FUNCTION_BLOCK "FB_PowerOn"   // FB462, SCL
{ S7_Optimized_Access := 'TRUE' }
// stored: AutoNumber false, MemoryReserve 100, SetENOAutomatically false
   VAR
      sMachinePower : Bool;
      sMachineReadySoft : Bool;
      sOkForPowerON : Bool;
      sTimeMachineReadyDelay { S7_SetPoint := 'True'} : TON_TIME;
      sDelayPowerOFF { S7_SetPoint := 'True'} : TON_TIME;
      sDelayPowerON_1 { S7_SetPoint := 'True'} : TON_TIME;
      sDelayPowerON_2 { S7_SetPoint := 'True'} : TON_TIME;
      sX_AxisBrakeRelease { S7_SetPoint := 'True'} : Bool;
      sY_AxisBrakeRelease : Bool;
      sB_AxisBrakeRelease : Bool;
   END_VAR
   VAR CONSTANT
      TIME_MACHINE_IN_DELAY : Time := T#2S;   // Output short pulse blinking
   END_VAR
BEGIN
   REGION Description header 
       //==================================================================================
       // POSALUX Swiss SA / (C) Copyright 2024
       //----------------------------------------------------------------------------------
       // Title: Power de la machine
       // Comment/Function: 
       //  A revoir le power des differents elements
       // Author: Gowsigan SRITHARAN
       // Engineering: TIA Portal v17
       //----------------------------------------------------------------------------------
       // Change log table:
       // Version  | Date     | Expert in charge | Changes applied
       // ---------|----------|------------------|------------------------------------
       // 00.00.01 | 20241120 | GSR              | First released version
       // ==================================================================================
   END_REGION

   REGION General Circuit breaker
       IF NOT "DB_DigitalInputs".sBreakerCtrl.sSWStatus THEN
           "LBP_AlarmMsgs".UserA[0].A70UUxx[3] := TRUE;
       END_IF;
   END_REGION

   REGION Operating counter
       "DB_DigitalOutputs".sOperatingCounter.sSWStatus :=
       ("LBP_Chan1".E_ProgRunning
       OR "LBP_Chan1".E_ProgWait)
       AND "LBP_ModeGroup".E_AUTO;
   END_REGION

   REGION Axis power requested
       #sOkForPowerON := "LBP_NC".E_NCKready AND "LBP_NC".E_DrivesInCylOp AND "DB_DataFromSafety".EmergencyStop AND NOT "DB_Alarms".sAlarmsLevel5 AND NOT "DB_Alarms".sAlarmsLevel6;

       IF #sOkForPowerON AND "DB_McpKeyboardSignals".sPowerON.sKeySWPositiveFront THEN
           #sMachinePower := TRUE;
       END_IF;

       IF  "DB_McpKeyboardSignals".sPowerOFF.sKeySWNegativeFront
           OR "DB_Machineshutdown_UPS".sShutDownPower
           OR "DB_Alarms".sAlarmsLevel5
           OR NOT "DB_DataFromSafety".EmergencyStop THEN
           #sMachinePower := FALSE;
       END_IF;

   END_REGION

   REGION Axis power output and waiting machine ready
       #sDelayPowerOFF(IN := NOT "LBP_NC".E_611Dready AND NOT #sMachinePower,
                       PT := T#1s);

       #sDelayPowerON_1(IN := "DB_DigitalOutputs".sInfeedON.sSWStatus,
                        PT := t#2s);
       #sDelayPowerON_2(IN := "DB_DigitalOutputs".sAxisActivation.sSWStatus,
                        PT := t#2s);
       IF #sMachinePower THEN
           "DB_DigitalOutputs".sInfeedON.sSWStatus := TRUE;
           IF #sDelayPowerON_1.Q THEN
               "DB_DigitalOutputs".sAxisActivation.sSWStatus := TRUE;
           END_IF;
           IF #sDelayPowerON_2.Q THEN

               "DB_DigitalOutputs".sAxis2_PowerContactor.sSWStatus  := TRUE;
               "DB_DigitalOutputs".sXY_AxisPowerContactor.sSWStatus := TRUE;
               "DB_DigitalOutputs".sBus60V_PowerContactor.sSWStatus := TRUE;
           END_IF;
       ELSE
           "DB_DigitalOutputs".sAxisActivation.sSWStatus := FALSE;

           IF #sDelayPowerOFF.Q THEN
               "DB_DigitalOutputs".sAxis2_PowerContactor.sSWStatus  := FALSE;
               "DB_DigitalOutputs".sXY_AxisPowerContactor.sSWStatus := FALSE;
               "DB_DigitalOutputs".sBus60V_PowerContactor.sSWStatus := FALSE;
               "DB_DigitalOutputs".sInfeedON.sSWStatus := FALSE;
           END_IF;
       END_IF;

       #sMachineReadySoft := "LBP_NC".E_611Dready;
   END_REGION

   REGION Machine in delay
       #sTimeMachineReadyDelay.TON(IN := #sMachineReadySoft,
                                   PT := #TIME_MACHINE_IN_DELAY);
   END_REGION

   REGION LED Machine ready start
       "DB_McpKeyboardSignals".sPowerON.sLedSWStatus :=
       (NOT #sMachinePower AND #sOkForPowerON AND "Clock_0.5Hz")
       OR (NOT #sTimeMachineReadyDelay.Q AND #sMachinePower AND "Clock_2Hz")
       OR #sTimeMachineReadyDelay.Q AND #sMachineReadySoft;
   END_REGION

   REGION Axis Brake
       // X Axis Brake Activation
       "DB_DigitalOutputs".sX_AxisBrakeActivation.sSWStatus := (("LBP_Axis01_X".E_AxisReady
       AND "LBP_Axis01_X".E_MotOK
       AND "LBP_Axis01_X".E_PulseEnable)
       OR #sX_AxisBrakeRelease);

       // Y Axis Brake Activation    
       "DB_DigitalOutputs".sY_AxisBrakeActivation.sSWStatus := (("LBP_Axis02_Y".E_AxisReady
       AND "LBP_Axis02_Y".E_MotOK
       AND "LBP_Axis02_Y".E_PulseEnable)
       OR #sY_AxisBrakeRelease);

       // B Axis Brake Activation   
       "DB_DigitalOutputs".sB_AxisBrakeRelease.sSWStatus := ("LBP_Axis04_B".E_AxisReady
       AND "LBP_Axis05_U1".E_MotOK
       AND "LBP_Axis05_U1".E_PulseEnable)
       OR #sB_AxisBrakeRelease;

       // Axis feed stop
       "LBP_AlarmMsgs".AxisA[1].AAFdStop60AAxx[0] := NOT "DB_DigitalOutputs".sX_AxisBrakeActivation.sSWStatus;     // X Axis
       "LBP_AlarmMsgs".AxisA[2].AAFdStop60AAxx[0] := NOT "DB_DigitalOutputs".sY_AxisBrakeActivation.sSWStatus;     // Y Axis
       "LBP_AlarmMsgs".AxisA[4].AAFdStop60AAxx[0] := NOT "DB_DigitalOutputs".sB_AxisBrakeRelease.sSWStatus;        // B Axis
   END_REGION
END_FUNCTION_BLOCK

FUNCTION_BLOCK "FB_Maintenances"   // FB473, SCL
{ S7_Optimized_Access := 'TRUE' }
// stored: AutoNumber false, MemoryReserve 100, SetENOAutomatically false
   VAR
      sCheckMachine : "FB_Maintenance";   // Message: Check Laser optical path (84h)
      sReplaceAirConditioningFilter { S7_SetPoint := 'True'} : "FB_Maintenance";   // Message: Clean the fairing (200 h)
      sMachineCooling_ReplaceWaterFilter { S7_SetPoint := 'True'} : "FB_Maintenance";   // Message: Clean the sheet metal (200 h)
      sTermotekChiller_ChangeFilterAndWater { S7_SetPoint := 'True'} : "FB_Maintenance";   // Message: Clean the screens (200 h)
      sCheckSafetySystem { S7_SetPoint := 'True'} : "FB_Maintenance";   // Message: Check the machine (200 h)
      sReplaceTipShellPeekGripper { S7_SetPoint := 'True'} : "FB_Maintenance";   // Message: Clean the clamping (200 h)
      sReplaceFiltersVacuumLoadingUnloading { S7_SetPoint := 'True'} : "FB_Maintenance";   // Message: Check the filter of the Laser power unit (2000 h)
      sReplaceFiltersVacuumGenerator { S7_SetPoint := 'True'} : "FB_Maintenance";   // Message: Check the safety systems (2000 h)
      sReplaceFilterAirDryer { S7_SetPoint := 'True'} : "FB_Maintenance";   // Message: Grease the X axis (1 y)
      sReplace5umFilter { S7_SetPoint := 'True'} : "FB_Maintenance";   // Message: Grease the Y axis (1 y)
      sReplace01umFilter { S7_SetPoint := 'True'} : "FB_Maintenance";   // Message: Check the water level of the TERMOTEK cooler (24 h)
      sReplaceActiveCarbonFilter { S7_SetPoint := 'True'} : "FB_Maintenance";   // Message: Clean the grid of the TERMOTEK cooler (24 h)
      sUTLExtraction_ReplaceParticleFilter { S7_SetPoint := 'True'} : "FB_Maintenance";   // Message: Check the operation of the condensate drain (24 h)
      sUTLExtraction_ReplaceFilterCassetteAndActiveCarbonFilter { S7_SetPoint := 'True'} : "FB_Maintenance";   // Message: Check the dew point under pressure (24 h)
      sReplaceSealOnSas { S7_SetPoint := 'True'} : "FB_Maintenance";   // Message: Clean the grid of the air dryer (24 h)
      sGreaseAxes { S7_SetPoint := 'True'} : "FB_Maintenance";   // Message: Replace the line filter of the air dryer (600 h)
      sMaintenance_16 { S7_SetPoint := 'True'} : "FB_Maintenance";   // Message: Replace 5 µm filter cartridge (600 h)
      sMaintenance_17 { S7_SetPoint := 'True'} : "FB_Maintenance";   // Message: Replace 0.01 µm filter cartridge (600 h)
      sMaintenance_18 { S7_SetPoint := 'True'} : "FB_Maintenance";   // Message: Replace the particles filter of the suction system (1000 h)
      sMaintenance_19 { S7_SetPoint := 'True'} : "FB_Maintenance";   // Message: Replace the filtration cassette AND the actived carbon of the suction system (1000 h)
      sMaintenance_20 { S7_SetPoint := 'True'} : "FB_Maintenance";   // Message: Replace the air conditioning filter (1000 h)
      sMaintenance_21 { S7_SetPoint := 'True'} : "FB_Maintenance";   // Message: Replace the TERMOTEK cooler filter (2000 h)
      sMaintenance_22 { S7_SetPoint := 'True'} : "FB_Maintenance";   // Message: Replace the water of the TERMOTEK cooler (2000 h)
      sMaintenance_23 { S7_SetPoint := 'True'} : "FB_Maintenance";   // Message: Spare
      sMaintenance_24 { S7_SetPoint := 'True'} : "FB_Maintenance";   // Message: Spare
      sMaintenance_25 { S7_SetPoint := 'True'} : "FB_Maintenance";   // Message: Spare
      sMaintenance_26 { S7_SetPoint := 'True'} : "FB_Maintenance";   // Message: Spare
      sMaintenance_27 { S7_SetPoint := 'True'} : "FB_Maintenance";   // Message: Spare
      sMaintenance_28 { S7_SetPoint := 'True'} : "FB_Maintenance";   // Message: Spare
      sMaintenance_29 { S7_SetPoint := 'True'} : "FB_Maintenance";   // Message: Spare
      sMaintenance_30 { S7_SetPoint := 'True'} : "FB_Maintenance";   // Message: Spare
      sMaintenance_31 { S7_SetPoint := 'True'} : "FB_Maintenance";   // Message: Spare
      sMaintenance_32 { S7_SetPoint := 'True'} : "FB_Maintenance";   // Message: Spare
      sMaintenance_33 { S7_SetPoint := 'True'} : "FB_Maintenance";   // Message: Spare
      sMaintenance_34 { S7_SetPoint := 'True'} : "FB_Maintenance";   // Message: Spare
      sMaintenance_35 { S7_SetPoint := 'True'} : "FB_Maintenance";   // Message: Spare
      sMaintenance_36 { S7_SetPoint := 'True'} : "FB_Maintenance";   // Message: Spare
      sMaintenance_37 { S7_SetPoint := 'True'} : "FB_Maintenance";   // Message: Spare
      sMaintenance_38 { S7_SetPoint := 'True'} : "FB_Maintenance";   // Message: Spare
      sMaintenance_39 { S7_SetPoint := 'True'} : "FB_Maintenance";   // Message: Spare
      sMaintenance_40 { S7_SetPoint := 'True'} : "FB_Maintenance";   // Message: Spare
      sMaintenance_41 { S7_SetPoint := 'True'} : "FB_Maintenance";   // Message: Spare
      sMaintenance_42 { S7_SetPoint := 'True'} : "FB_Maintenance";   // Message: Spare
      sMaintenance_43 { S7_SetPoint := 'True'} : "FB_Maintenance";   // Message: Spare
      sMaintenance_44 { S7_SetPoint := 'True'} : "FB_Maintenance";   // Message: Spare
      sMaintenance_45 { S7_SetPoint := 'True'} : "FB_Maintenance";   // Message: Spare
      sMaintenance_46 { S7_SetPoint := 'True'} : "FB_Maintenance";   // Message: Spare
      sMaintenance_47 { S7_SetPoint := 'True'} : "FB_Maintenance";   // Message: Spare
      sMaintenance_48 { S7_SetPoint := 'True'} : "FB_Maintenance";   // Message: Spare
      sMaintenance_49 { S7_SetPoint := 'True'} : "FB_Maintenance";   // Message: Spare
      sMaintenance_50 { S7_SetPoint := 'True'} : "FB_Maintenance";   // Message: Spare
      sMaintenance_51 { S7_SetPoint := 'True'} : "FB_Maintenance";   // Message: Spare
      sMaintenance_52 { S7_SetPoint := 'True'} : "FB_Maintenance";   // Message: Spare
      sMaintenance_53 { S7_SetPoint := 'True'} : "FB_Maintenance";   // Message: Spare
      sMaintenance_54 { S7_SetPoint := 'True'} : "FB_Maintenance";   // Message: Spare
      sMaintenance_55 { S7_SetPoint := 'True'} : "FB_Maintenance";   // Message: Spare
      sMaintenance_56 { S7_SetPoint := 'True'} : "FB_Maintenance";   // Message: Spare
      sMaintenance_57 { S7_SetPoint := 'True'} : "FB_Maintenance";   // Message: Spare
      sMaintenance_58 { S7_SetPoint := 'True'} : "FB_Maintenance";   // Message: Spare
      sMaintenance_59 { S7_SetPoint := 'True'} : "FB_Maintenance";   // Message: Spare
      sMaintenance_60 { S7_SetPoint := 'True'} : "FB_Maintenance";   // Message: Spare
      sMaintenance_61 { S7_SetPoint := 'True'} : "FB_Maintenance";   // Message: Spare
      sMaintenance_62 { S7_SetPoint := 'True'} : "FB_Maintenance";   // Message: Spare
      sMaintenance_63 { S7_SetPoint := 'True'} : "FB_Maintenance";   // Message: Spare
   END_VAR
BEGIN
   REGION Description header 
       //==================================================================================
       // POSALUX Swiss SA / (C) Copyright 2024
       //----------------------------------------------------------------------------------
       // Title: Maintenance
       // Comment/Function: Liste des apparaeils à controler dans la Liste des équipements 
       //                   pour la maintenance préventive  
       //
       // Author: Gowsigan SRITHARAN
       // Engineering: TIA Portal v17
       //----------------------------------------------------------------------------------
       // Change log table:
       // Version  | Date     | Expert in charge | Changes applied
       // ---------|----------|------------------|------------------------------------
       // 00.00.01 | 20250912 | WFA              | First released version
       // ==================================================================================
   END_REGION

   REGION 200 hours
           // Check the machine
           #sCheckMachine(iIncrementEnable := "LBP_Chan1".E_ProgRunning,
                          iID := 101,
                          ioOPC := "DB_OPC_Maintenance".Tasks[1],
                          ioAlarm := "LBP_AlarmMsgs".UserA[30].A70UUxx[00],
                          ioWarning := "LBP_AlarmMsgs".UserA[30].A70UUxx[32]);
      END_REGION

      REGION 1000 hours
           // Replace the air conditioning filter
           #sReplaceAirConditioningFilter(iIncrementEnable := "LBP_Chan1".E_ProgRunning,
                                          iID := 201,
                                          ioOPC := "DB_OPC_Maintenance".Tasks[2],
                                          ioAlarm := "LBP_AlarmMsgs".UserA[30].A70UUxx[01],
                                          ioWarning := "LBP_AlarmMsgs".UserA[30].A70UUxx[33]);

           // Machine cooling: replace water filter
           #sMachineCooling_ReplaceWaterFilter(iIncrementEnable := "LBP_Chan1".E_ProgRunning,
                                               iID := 202,
                                               ioOPC := "DB_OPC_Maintenance".Tasks[3],
                                               ioAlarm := "LBP_AlarmMsgs".UserA[30].A70UUxx[02],
                                               ioWarning := "LBP_AlarmMsgs".UserA[30].A70UUxx[34]);
      END_REGION

      REGION 2000 hours
          // Termotek chiller: change filter and water
          #sTermotekChiller_ChangeFilterAndWater(iIncrementEnable := "LBP_Chan1".E_ProgRunning,
                                                 iID := 301,
                                                 ioOPC := "DB_OPC_Maintenance".Tasks[4],
                                                 ioAlarm := "LBP_AlarmMsgs".UserA[30].A70UUxx[03],
                                                 ioWarning := "LBP_AlarmMsgs".UserA[30].A70UUxx[35]);

           // Check the safety system
           #sCheckSafetySystem(iIncrementEnable := "LBP_Chan1".E_ProgRunning,
                               iID := 302,
                               ioOPC := "DB_OPC_Maintenance".Tasks[5],
                               ioAlarm := "LBP_AlarmMsgs".UserA[30].A70UUxx[04],
                               ioWarning := "LBP_AlarmMsgs".UserA[30].A70UUxx[36]);

           // Replace the tip-shell PEEK gripper
           #sReplaceTipShellPeekGripper(iIncrementEnable := "LBP_Chan1".E_ProgRunning,
                                        iID := 303,
                                        ioOPC := "DB_OPC_Maintenance".Tasks[6],
                                        ioAlarm := "LBP_AlarmMsgs".UserA[30].A70UUxx[05],
                                        ioWarning := "LBP_AlarmMsgs".UserA[30].A70UUxx[37]);
      END_REGION

      REGION 3000 hours
           // Replace the filters for the vacuum of the loading/unloading
           #sReplaceFiltersVacuumLoadingUnloading(iIncrementEnable := "LBP_Chan1".E_ProgRunning,
                                                  iID := 401,
                                                  ioOPC := "DB_OPC_Maintenance".Tasks[7],
                                                  ioAlarm := "LBP_AlarmMsgs".UserA[30].A70UUxx[06],
                                                  ioWarning := "LBP_AlarmMsgs".UserA[30].A70UUxx[38]);

           // Replace the filters of the vacuum generator VADM
           #sReplaceFiltersVacuumGenerator(iIncrementEnable := "LBP_Chan1".E_ProgRunning,
                                           iID := 402,
                                           ioOPC := "DB_OPC_Maintenance".Tasks[8],
                                           ioAlarm := "LBP_AlarmMsgs".UserA[30].A70UUxx[07],
                                           ioWarning := "LBP_AlarmMsgs".UserA[30].A70UUxx[39]);
      END_REGION

      REGION 4000 hours
           // Replace the fine filter of the air dryer
           #sReplaceFilterAirDryer(iIncrementEnable := "LBP_Chan1".E_ProgRunning,
                                   iID := 501,
                                   ioOPC := "DB_OPC_Maintenance".Tasks[9],
                                   ioAlarm := "LBP_AlarmMsgs".UserA[30].A70UUxx[08],
                                   ioWarning := "LBP_AlarmMsgs".UserA[30].A70UUxx[40]);

           // Replace the 5 μm filter
           #sReplace5umFilter(iIncrementEnable := "LBP_Chan1".E_ProgRunning,
                              iID := 502,
                              ioOPC := "DB_OPC_Maintenance".Tasks[10],
                              ioAlarm := "LBP_AlarmMsgs".UserA[30].A70UUxx[09],
                              ioWarning := "LBP_AlarmMsgs".UserA[30].A70UUxx[41]);

          // Replace the 0.1 μm filter
         #sReplace01umFilter(iIncrementEnable := "LBP_Chan1".E_ProgRunning,
                             iID := 503,
                             ioOPC := "DB_OPC_Maintenance".Tasks[11],
                             ioAlarm := "LBP_AlarmMsgs".UserA[30].A70UUxx[10],
                             ioWarning := "LBP_AlarmMsgs".UserA[30].A70UUxx[42]);

           // Replace the active carbon filter
           #sReplaceActiveCarbonFilter(iIncrementEnable := "LBP_Chan1".E_ProgRunning,
                                       iID := 504,
                                       ioOPC := "DB_OPC_Maintenance".Tasks[12],
                                       ioAlarm := "LBP_AlarmMsgs".UserA[30].A70UUxx[11],
                                       ioWarning := "LBP_AlarmMsgs".UserA[30].A70UUxx[43]);

           // UTL extraction: replace particle filter
           #sUTLExtraction_ReplaceParticleFilter(iIncrementEnable := "LBP_Chan1".E_ProgRunning,
                                                 iID := 505,
                                                 ioOPC := "DB_OPC_Maintenance".Tasks[13],
                                                 ioAlarm := "LBP_AlarmMsgs".UserA[30].A70UUxx[12],
                                                 ioWarning := "LBP_AlarmMsgs".UserA[30].A70UUxx[44]);

           // UTL extraction: replace filter cassette and active carbon filter
           #sUTLExtraction_ReplaceFilterCassetteAndActiveCarbonFilter(iIncrementEnable := "LBP_Chan1".E_ProgRunning,
                                                                      iID := 506,
                                                                      ioOPC := "DB_OPC_Maintenance".Tasks[14],
                                                                      ioAlarm := "LBP_AlarmMsgs".UserA[30].A70UUxx[13],
                                                                      ioWarning := "LBP_AlarmMsgs".UserA[30].A70UUxx[45]);

      END_REGION

      REGION 6000 hours
           // Replace the seal on the air lock door (SAS)
           #sReplaceSealOnSas(iIncrementEnable := "LBP_Chan1".E_ProgRunning,
                              iID := 601,
                              ioOPC := "DB_OPC_Maintenance".Tasks[15],
                              ioAlarm := "LBP_AlarmMsgs".UserA[30].A70UUxx[14],
                              ioWarning := "LBP_AlarmMsgs".UserA[30].A70UUxx[46]);

           // Grease the axes
           #sGreaseAxes(iIncrementEnable := "LBP_Chan1".E_ProgRunning,
                        iID := 602,
                        ioOPC := "DB_OPC_Maintenance".Tasks[16],
                        ioAlarm := "LBP_AlarmMsgs".UserA[30].A70UUxx[15],
                        ioWarning := "LBP_AlarmMsgs".UserA[30].A70UUxx[47]);
      END_REGION
END_FUNCTION_BLOCK

FUNCTION_BLOCK "FB_Maintenance"   // FB471, SCL
{ S7_Optimized_Access := 'TRUE' }
// stored: AutoNumber false, MemoryReserve 100, SetENOAutomatically false
   VAR_INPUT
      iIncrementEnable { ExternalAccessible := 'False'; ExternalVisible := 'False'; ExternalWritable := 'False'} : Bool;
      iID { ExternalAccessible := 'False'; ExternalVisible := 'False'; ExternalWritable := 'False'} : Int;
   END_VAR
   VAR_IN_OUT
      ioOPC : "UDT_OPC_Maintenance";
      ioAlarm { ExternalAccessible := 'False'; ExternalVisible := 'False'; ExternalWritable := 'False'} : Bool;   // Alarme (100% atteint)
      ioWarning { ExternalAccessible := 'False'; ExternalVisible := 'False'; ExternalWritable := 'False'} : Bool;   // Avertissement (80% atteint)
   END_VAR
   VAR
      sElement { ExternalAccessible := 'False'; ExternalVisible := 'False'; ExternalWritable := 'False'} : "UDT_MaintenanceElement";
   END_VAR
   VAR_TEMP
      tUsagePercent : Real;
      tAdjustedIncrement : Bool;
   END_VAR
BEGIN
   REGION Description header 
       //==================================================================================
       // POSALUX Swiss SA / (C) Copyright 2024
       //----------------------------------------------------------------------------------
       // Title: Gestion_Temps_Fonctionnement
       // Comment/Function: Cette fonction  assure le suivi du temps de fonctionnement
       //                   des équipements et génère des alertes basées sur
       //                   leur utilisation. Elle incrémente le temps de fonctionnement
       //                   selon l'unité définie (minute, heure, jour), calcule le
       //                   pourcentage d'utilisation par rapport à un seuil d'alarme, et
       //                   gère les avertissements et alarmes en fonction de ce pourcentage
       //
       // Author: Gowsigan SRITHARAN
       // Engineering: TIA Portal v17
       //----------------------------------------------------------------------------------
       // Change log table:
       // Version  | Date     | Expert in charge | Changes applied
       // ---------|----------|------------------|------------------------------------
       // 00.00.01 | 20241120 | GSR              | First released version
       // ---------|----------|------------------|------------------------------------
       // 01.01.01 | 20241219 | FMI              | Utilisation d'un flanc montant du clock1Hz pour compter en secondes
       // ==================================================================================
   END_REGION

   REGION Incrementation du temps en secondes
       IF "DB_Impulsion".sRT_Clock_1Hz.Q AND #iIncrementEnable THEN
           #sElement.RunTimeSec := #sElement.RunTimeSec + 1;
       END_IF;
   END_REGION

   REGION Incrementation du temps en fonction du type unité
       CASE #sElement.TimeUnit OF
           0:
               #sElement.RunTime := #sElement.RunTimeSec / 60.0;     // Affichage runtime en minutes
           1:
               #sElement.RunTime := #sElement.RunTimeSec / 3600.0;   // Affichage runtime en heures
           2:
               #sElement.RunTime := #sElement.RunTimeSec / 86400.0;  // Affichage runtime en jours
       END_CASE;

   END_REGION

   REGION Gestion des warnings et alarmes    
       // Définir l'état de l'alarme et des avertissements en fonction du pourcentage d'utilisation
       #ioAlarm   := #sElement.RunTime >= #sElement.AlarmThreshold;                      // Alarme si utilisation atteint ou dépasse le seuil d'alarme
       #ioWarning := #sElement.RunTime >= #sElement.WarningThreshold AND NOT #ioAlarm;   // Avertissement si utilisation dépasse le seuil d'avertissement sans alarme active
   END_REGION

   REGION OPC Communication
       #ioOPC.Elapsed := #sElement.RunTime;
       #ioOPC.WarningThreshold := #sElement.WarningThreshold;
       #ioOPC.Period := #sElement.AlarmThreshold;
       #ioOPC.Id := #iID;
       #sElement.ResetRunTime :=#ioOPC.Reset;
       #ioOPC.Reset := FALSE;
   END_REGION

   REGION Reset du compteur
       IF #sElement.ResetRunTime THEN
           #sElement.RunTimeSec := 0;       // Reset du compteur de temps de fonctionnement
           #sElement.ResetRunTime := FALSE;
       END_IF;
   END_REGION
END_FUNCTION_BLOCK

FUNCTION_BLOCK "FB_Temperature"   // FB490, SCL
{ S7_Optimized_Access := 'TRUE' }
// stored: AutoNumber false, MemoryReserve 100, SetENOAutomatically false
   VAR
      sPIDRestart : Bool;
      sPIDHoldI : Bool;
      sXAxisWarning : Real := 50.0;
      sPIDClimOut : Real;
      sP : Real := -100.0;
      sI : Time := T#10D;
      sD : Time := T#12S;
      sTimeOutFlowChiller : TON_TIME;
      sTimeOutLevelChiller { S7_SetPoint := 'True'} : TON_TIME;
      sTimeOutChillerGood : TON_TIME;
      sTimeOutCooling : TON_TIME;
      sTemperature_X_PT1000 { S7_SetPoint := 'True'} : "FB_AnalogInputThreshold";
      sTemperature_Y_PT1000 { S7_SetPoint := 'True'} : "FB_AnalogInputThreshold";
      sAmbiantTemperature { S7_SetPoint := 'True'} : "FB_AnalogInputThreshold";
      sMachineTemperature { S7_SetPoint := 'True'} : "FB_AnalogInputThreshold";
      sCabinetTemperatureMeasure { S7_SetPoint := 'True'} : "FB_AnalogInputThreshold";
      sColdWaterTemperatureInput { S7_SetPoint := 'True'} : "FB_AnalogInputThreshold";
      sColdWaterTemperatureOutput { S7_SetPoint := 'True'} : "FB_AnalogInputThreshold";
      sTemperatureCooling { S7_SetPoint := 'True'} : "FB_AnalogInputThreshold";
   END_VAR
   VAR_TEMP
      tSetPointCheck : Real;
      tDataAction : "AnalogInAction_DT";
   END_VAR
   VAR CONSTANT
      ALARM_PTC : Real := 110.0;
      TIME_OUT_COOLING : Time := T#5S;
   END_VAR
BEGIN
   REGION Description header 
       //==================================================================================
       // POSALUX Swiss SA / (C) Copyright 2024
       //----------------------------------------------------------------------------------
       // Title: Temperatures management
       // Comment/Function: 
       //
       // Author: Gowsigan SRITHARAN
       // Engineering: TIA Portal v17
       //----------------------------------------------------------------------------------
       // Change log table:
       // Version  | Date     | Expert in charge | Changes applied
       // ---------|----------|------------------|------------------------------------
       // 00.00.01 | 20241120 | GSR              | First released version
       // ==================================================================================
   END_REGION

   REGION Ambiant temperature (externe)  
       #sAmbiantTemperature(iActualValue := "DB_AnalogInputs".sAmbiantTemperature.sSWRealValue,
                            iStartDelay := TRUE,
                            ioAlarmMin := "LBP_AlarmMsgs".UserA[06].A70UUxx[04],
                            ioWarningMin := "LBP_AlarmMsgs".UserA[07].A70UUxx[04],
                            ioWarningMax := "LBP_AlarmMsgs".UserA[07].A70UUxx[05],
                            ioAlarmMax := "LBP_AlarmMsgs".UserA[06].A70UUxx[05],
                            oDataAction => "DB_AnalogInputAction".Ambiant_Temperature,
                            iDataPLC := "DB_AnalogInputDataPLC".Ambiant_Temperature,
                            iDataHMI := "DB_AnalogInputDataHMI".Ambiant_Temperature);
   END_REGION

   REGION Water input  
       #sColdWaterTemperatureInput(iActualValue := "DB_AnalogInputs".sCold_WaterTemperatureInput.sSWRealValue,
                                   iStartDelay := TRUE,
                                   ioAlarmMin := "LBP_AlarmMsgs".UserA[06].A70UUxx[08],
                                   ioWarningMin := "LBP_AlarmMsgs".UserA[07].A70UUxx[08],
                                   ioWarningMax := "LBP_AlarmMsgs".UserA[07].A70UUxx[09],
                                   ioAlarmMax := "LBP_AlarmMsgs".UserA[06].A70UUxx[09],
                                   oDataAction => "DB_AnalogInputAction".Cold_Water_Temperature_Input,
                                   iDataPLC := "DB_AnalogInputDataPLC".Cold_Water_Temperature_Input,
                                   iDataHMI := "DB_AnalogInputDataHMI".Cold_Water_Temperature_Input);
   END_REGION

   REGION Cooling On
       "DB_DigitalOutputs".sCoolingStart.sSWStatus := "DB_PowerOn".sMachineReadySoft;
   END_REGION ;

   REGION Cooling alarm
       #sTimeOutCooling(IN := "DB_PowerOn".sTimeMachineReadyDelay.Q AND NOT "DB_DigitalInputs".sCoolingOK.sSWStatus,
                        PT := #TIME_OUT_COOLING,
                        Q => "LBP_AlarmMsgs".UserA[4].A70UUxx[10]);
   END_REGION

   REGION Water output   
       #sColdWaterTemperatureOutput(iActualValue := "DB_AnalogInputs".sCold_WaterTemperatureOutput.sSWRealValue,
                                    iStartDelay := TRUE,
                                    ioAlarmMin := "LBP_AlarmMsgs".UserA[06].A70UUxx[10],
                                    ioWarningMin := "LBP_AlarmMsgs".UserA[07].A70UUxx[10],
                                    ioWarningMax := "LBP_AlarmMsgs".UserA[07].A70UUxx[11],
                                    ioAlarmMax := "LBP_AlarmMsgs".UserA[06].A70UUxx[11],
                                    oDataAction => "DB_AnalogInputAction".Cold_Water_Temperature_Output,
                                    iDataPLC := "DB_AnalogInputDataPLC".Cold_Water_Temperature_Output,
                                    iDataHMI := "DB_AnalogInputDataHMI".Cold_Water_Temperature_Output);
   END_REGION

   REGION X Axis temperature check
       #sTemperature_X_PT1000(iActualValue := "DB_AnalogInputs".sX_AxisTemperaturePT1000.sSWRealValue,
                              iStartDelay := TRUE,
                              ioAlarmMin := "LBP_AlarmMsgs".UserA[06].A70UUxx[00],
                              ioWarningMin := "LBP_AlarmMsgs".UserA[07].A70UUxx[00],
                              ioWarningMax := "LBP_AlarmMsgs".UserA[07].A70UUxx[01],
                              ioAlarmMax := "LBP_AlarmMsgs".UserA[06].A70UUxx[01],
                              oDataAction => "DB_AnalogInputAction".X_Axis_Temperature_PT1000,
                              iDataPLC := "DB_AnalogInputDataPLC".X_Axis_Temperature_PT1000,
                              iDataHMI := "DB_AnalogInputDataHMI".X_Axis_Temperature_PT1000);

       // Temperature_X_PTC
       // PTC used as a temperature threshold rather than a measurement
       IF "DB_AnalogInputs".sX_AxisTemperaturePTC.iValueHW.%X0 OR "DB_AnalogInputs".sX_AxisTemperaturePTC.iValueHW.%X2 THEN
           "LBP_AlarmMsgs".UserA[06].A70UUxx[23] := TRUE;
       END_IF;
   END_REGION

   REGION Y Axis temperature check
       #sTemperature_Y_PT1000(iActualValue := "DB_AnalogInputs".sY_AxisTemperaturePT1000.sSWRealValue,
                              iStartDelay := TRUE,
                              ioAlarmMin := "LBP_AlarmMsgs".UserA[06].A70UUxx[02],
                              ioWarningMin := "LBP_AlarmMsgs".UserA[07].A70UUxx[02],
                              ioWarningMax := "LBP_AlarmMsgs".UserA[07].A70UUxx[03],
                              ioAlarmMax := "LBP_AlarmMsgs".UserA[06].A70UUxx[03],
                              oDataAction => "DB_AnalogInputAction".Y_Axis_Temperature_PT1000,
                              iDataPLC := "DB_AnalogInputDataPLC".Y_Axis_Temperature_PT1000,
                              iDataHMI := "DB_AnalogInputDataHMI".Y_Axis_Temperature_PT1000);

       // Temperature_Y_PTC
       // PTC used as a temperature threshold rather than a measurement
       IF "DB_AnalogInputs".sY_AxisTemperaturePTC.iValueHW.%X0 OR "DB_AnalogInputs".sY_AxisTemperaturePTC.iValueHW.%X2 THEN
           "LBP_AlarmMsgs".UserA[06].A70UUxx[25] := TRUE;
       END_IF;
   END_REGION

   REGION Electrical Cabinet
       #sCabinetTemperatureMeasure(iActualValue := "DB_AnalogInputs".sCabinetTemperature.sSWRealValue,
                                   iStartDelay := TRUE,
                                   ioAlarmMin := "LBP_AlarmMsgs".UserA[06].A70UUxx[52],
                                   ioWarningMin := "LBP_AlarmMsgs".UserA[07].A70UUxx[52],
                                   ioWarningMax := "LBP_AlarmMsgs".UserA[07].A70UUxx[53],
                                   ioAlarmMax := "LBP_AlarmMsgs".UserA[06].A70UUxx[53],
                                   oDataAction => "DB_AnalogInputAction".Cabinet_Temperature,
                                   iDataPLC := "DB_AnalogInputDataPLC".Cabinet_Temperature,
                                   iDataHMI := "DB_AnalogInputDataHMI".Cabinet_Temperature);

       IF "DB_DigitalInputs".sCabinetTemperatureCtrl.sSWStatus THEN
            "LBP_AlarmMsgs".UserA[0].A70UUxx[4] := TRUE;
        END_IF;
    END_REGION

    REGION Machine management temperature (interieur)
        #sMachineTemperature(iActualValue := "DB_AnalogInputs".sMachineTemperature.sSWRealValue,
                             iStartDelay := TRUE,
                             ioAlarmMin := "LBP_AlarmMsgs".UserA[06].A70UUxx[06],
                             ioWarningMin := "LBP_AlarmMsgs".UserA[07].A70UUxx[06],
                             ioWarningMax := "LBP_AlarmMsgs".UserA[07].A70UUxx[07],
                             ioAlarmMax := "LBP_AlarmMsgs".UserA[06].A70UUxx[07],
                             oDataAction => "DB_AnalogInputAction".Machine_Temperature,
                             iDataPLC := "DB_AnalogInputDataPLC".Machine_Temperature,
                             iDataHMI := "DB_AnalogInputDataHMI".Machine_Temperature);

        REGION Machine ventilator
            // Ventilator setpoint (from HMI) Forcing value under 0% OR over 100%
            IF "DB_HMISetting".CoolingVentilatorSetpoint < 0.0 THEN
                "DB_HMISetting".CoolingVentilatorSetpoint := 0.0;
            ELSIF "DB_HMISetting".CoolingVentilatorSetpoint > 100.0 THEN
                "DB_HMISetting".CoolingVentilatorSetpoint := 100.0;
            END_IF;

            IF "DB_DigitalOutputs".sXY_AxisPowerContactor.sSWStatus OR
                "DB_DigitalOutputs".sAxis2_PowerContactor.sSWStatus OR
                "DB_DigitalOutputs".sBus60V_PowerContactor.sSWStatus THEN
                "DB_AnalogOutputs".sVentilatorSetPoint.sSWRealValue := "DB_HMISetting".CoolingVentilatorSetpoint;
            ELSE
                "DB_AnalogOutputs".sVentilatorSetPoint.sSWRealValue := 0.0;
            END_IF;
        END_REGION

        REGION Check setpoint temperature machine
            #sTemperatureCooling(iActualValue := "DB_AnalogInputs".sClimTemperature.sSWRealValue,
                                 iStartDelay := TRUE,
                                 ioAlarmMin := "LBP_AlarmMsgs".UserA[06].A70UUxx[54],
                                 ioWarningMin := "LBP_AlarmMsgs".UserA[07].A70UUxx[54],
                                 ioWarningMax := "LBP_AlarmMsgs".UserA[07].A70UUxx[55],
                                 ioAlarmMax := "LBP_AlarmMsgs".UserA[06].A70UUxx[55],
                                 oDataAction => #tDataAction,
                                 iDataPLC := "DB_AnalogInputDataPLC".Clim_Temperature,
                                 iDataHMI := "DB_AnalogInputDataHMI".Clim_Temperature);
        END_REGION

        // REGION Machine temperature cooling PID WFA Déplacé dans OB30
        //     "CONT_C_Clim_DB"(COM_RST := #sPIDRestart,
        //                      MAN_ON := FALSE,
        //                      P_SEL := TRUE,
        //                      I_SEL := TRUE,
        //                      INT_HOLD := #sPIDHoldI,
        //                      D_SEL := TRUE,
        //                      CYCLE := T#1s,
        //                      SP_INT := "DB_HMISetting".TemperatureCoolingSetpoint,
        //                      PV_IN := "DB_AnalogInputs".sClimTemperature.sSWRealValue,
        //                      GAIN := #sP,
        //                      TI := #sI,
        //                      TD := #sD,
        //                      DEADB_W := 0.1,
        //                      LMN_HLM := 100,
        //                      LMN_LLM := 0,
        //                      LMN => "DB_AnalogOutputs".sPropValveClimSetPoint.sSWRealValue);
        // END_REGION
    END_REGION
END_FUNCTION_BLOCK

FUNCTION_BLOCK "FB_WarmUP"   // FB530, SCL
{ S7_Optimized_Access := 'TRUE' }
// stored: AutoNumber false, MemoryReserve 100, SetENOAutomatically false
   VAR
      sWarmUpTimer : Time;
      sLimitedWarmupTime : Bool;
      sUnlimitedWarmupTime : Bool;
      sActualWarmupTime : Time;
      sRemainingWarmupMinutes : Int;
      sDeltaTimeWarmup : Time;
      sLimitedWarmUP : TON_TIME;
      sStartWarmup { S7_SetPoint := 'True'} : Bool;
      sUnlimitedWarmUP : TON_TIME;
      sUnlimitedWarmUPCounter { S7_SetPoint := 'True'} : "FB_TimeCounter";
   END_VAR
   VAR CONSTANT
      WU_MIN : Int := 30;
   END_VAR
BEGIN
   REGION Description header 
       //==================================================================================
       // POSALUX Swiss SA / (C) Copyright 2024
       //----------------------------------------------------------------------------------
       // Title: Laser Warm-up
       // Comment/Function: 
       // This block manages the laser warm-up process. It includes functionality for both limited
       // and unlimited warm-up times.
       //
       // Author: [Gowsigan SRITHARAN]
       // Engineering: TIA Portal [version]
       //----------------------------------------------------------------------------------
       // Change log table:
       // Version  | Date     | Expert in charge | Changes applied
       // ---------|----------|------------------|------------------------------------
       // 00.00.01 | 20250224 | gsr              | First released version
       // 00.00.02 | 20250314 | wfa              | Modification unlimited timer
       // ==================================================================================
   END_REGION

   REGION Selection Warm-UP mode: limited or unlimited
       // Timer for unlimited Warm-UP detection
       #sUnlimitedWarmUP(IN := "DB_McpKeyboardSignals".sK14_WarmUp.sKeySWStatus OR "DB_HmiKeyboardSignals".sK14_WarmUp.sKeySWStatus,
                         PT := T#2s);

       // Warm-up mode selection logic
       IF ("DB_McpKeyboardSignals".sK14_WarmUp.sKeySWStatus OR "DB_HmiKeyboardSignals".sK14_WarmUp.sKeySWStatus) AND "LBP_ModeGroup".E_AUTO AND NOT #sUnlimitedWarmUP.Q THEN
           // Activate unlimited Warm-UP when key is initially pressed
           #sLimitedWarmupTime := FALSE;
           #sUnlimitedWarmupTime := TRUE;
           #sStartWarmup := TRUE;
       ELSIF "DB_McpKeyboardSignals".sK14_WarmUp.sKeySWStatus AND "DB_HmiKeyboardSignals".sK14_WarmUp.sKeySWStatus AND "LBP_ModeGroup".E_AUTO AND #sUnlimitedWarmUP.Q THEN
           // Switch to limited Warm-UP if key is held for 2 seconds
           #sLimitedWarmupTime := TRUE;
           #sUnlimitedWarmupTime := FALSE;
           #sStartWarmup := TRUE;
           #sWarmUpTimer := DINT_TO_TIME(DINT_TO_INT(#WU_MIN * 60 * 1000)); // Limited time in milliseconds
       ELSIF "DB_McpKeyboardSignals".sK14_WarmUp.sKeySWToggleStatus = FALSE AND "DB_HmiKeyboardSignals".sK14_WarmUp.sKeySWToggleStatus THEN
           #sLimitedWarmupTime := FALSE;
           #sUnlimitedWarmupTime := FALSE;
           #sStartWarmup := FALSE;
       END_IF;
   END_REGION

   REGION Warm-UP Counter (Unlimited Warm-Up)
       #sUnlimitedWarmUPCounter(iStart := #sUnlimitedWarmupTime AND ("LBP_Chan1".E_ProgRunning OR "LBP_Chan1".E_ProgWait OR "LBP_Chan1".E_ProgStop),
                                iReset := NOT "DB_McpKeyboardSignals".sK14_WarmUp.sKeySWToggleStatus AND NOT "DB_HmiKeyboardSignals".sK14_WarmUp.sKeySWToggleStatus);
   END_REGION ;

   REGION Warm-UP Timer  (Limited Warm-up)  
       // Start the Warm-UP timer
       #sLimitedWarmUP.TON(IN := #sLimitedWarmupTime AND ("LBP_Chan1".E_ProgRunning OR "LBP_Chan1".E_ProgWait OR "LBP_Chan1".E_ProgStop),
                           PT := #sWarmUpTimer);

       IF #sLimitedWarmUP.Q THEN
           "DB_McpKeyboardSignals".sK14_WarmUp.sKeySWToggleStatus := FALSE;
           "DB_HmiKeyboardSignals".sK14_WarmUp.sKeySWToggleStatus := FALSE;
       END_IF;
   END_REGION

   REGION Update NC inputs and MCP LED status
       "LBP_NC".A_Set_Inp34 := "DB_McpKeyboardSignals".sK14_WarmUp.sKeySWToggleStatus OR "DB_HmiKeyboardSignals".sK14_WarmUp.sKeySWToggleStatus;

       "DB_McpKeyboardSignals".sK14_WarmUp.sLedSWStatus :=
       "DB_McpKeyboardSignals".sK14_WarmUp.sKeySWToggleStatus
       AND (#sUnlimitedWarmupTime OR "Clock_2Hz");

       "DB_HmiKeyboardSignals".sK14_WarmUp.sLedSWStatus :=
       "DB_HmiKeyboardSignals".sK14_WarmUp.sKeySWToggleStatus
       AND (#sUnlimitedWarmupTime OR "Clock_2Hz");
   END_REGION

   REGION Display Remaining Time
       IF #sLimitedWarmupTime THEN
           // Display remaining time for limited warm-up
           "DB_HMIStatus".WarmUpTime := DINT_TO_REAL(TIME_TO_DINT(#sLimitedWarmUP.PT - #sLimitedWarmUP.ET)) / 1000.0;
       ELSIF #sUnlimitedWarmupTime THEN
           // Display elapsed time for unlimited warm-up
           "DB_HMIStatus".WarmUpTime := #sUnlimitedWarmUPCounter.ioSecondsCumul;
       ELSE
           // Reset display when conditions are not met
           "DB_HMIStatus".WarmUpTime := 0;
       END_IF;
   END_REGION

   REGION Warm-UP Message
       IF "LBP_ModeGroup".E_AUTO AND "LBP_NC".A_Set_Inp34 AND
           ("LBP_Chan1".E_ProgRunning OR "LBP_Chan1".E_ProgWait OR "LBP_Chan1".E_ProgStop) THEN
           "LBP_AlarmMsgs".UserA[0].A70UUxx[35] := TRUE;
       END_IF;
   END_REGION

   REGION Warm-UP Status
       "DB_HMIStatus".WarmUpOn := #sStartWarmup;
   END_REGION

   REGION Warm-UP Status To NC
       "DB_PLC_ISO_IHM".WarmUpOn := "DB_McpKeyboardSignals".sK14_WarmUp.sKeySWToggleStatus OR "DB_HmiKeyboardSignals".sK14_WarmUp.sKeySWToggleStatus;
   END_REGION
END_FUNCTION_BLOCK

FUNCTION_BLOCK "FB_FeedOverride"   // FB82, SCL
{ S7_Optimized_Access := 'TRUE' }
// stored: MemoryReserve 100, SetENOAutomatically false
   VAR_INPUT
      iA_FD_OR : Byte;
   END_VAR
   VAR_OUTPUT
      oFeedOverride : Byte;
   END_VAR
BEGIN
   REGION Description header 
       //==================================================================================
       // POSALUX Swiss SA / (C) Copyright 2026
       //----------------------------------------------------------------------------------
       // Title: FB_FeedObverride
       // Comment/Function: 
       // Author: Fabien WALDT
       // Engineering: TIA Portal v20
       //----------------------------------------------------------------------------------
       // Change log table:
       // Version  | Date     | Expert in charge | Changes applied
       // ---------|----------|------------------|-----------------------------------------
       // 00.00.01 | 20260309 | WFA              | First released version
       // =================================================================================
   END_REGION

   REGION Feed Ovr Value
       CASE #iA_FD_OR OF
           1:
               #oFeedOverride := 0;
           3:
               #oFeedOverride := 1;
           2:
               #oFeedOverride := 2;
           6:
               #oFeedOverride := 4;
           7:
               #oFeedOverride := 6;
           5:
               #oFeedOverride := 8;
           4:
               #oFeedOverride := 10;
           12:
               #oFeedOverride := 20;
           13:
               #oFeedOverride := 30;
           15:
               #oFeedOverride := 40;
           14:
               #oFeedOverride := 50;
           10:
               #oFeedOverride := 60;
           11:
               #oFeedOverride := 70;
           9:
               #oFeedOverride := 75;
           8:
               #oFeedOverride := 80;
           24:
               #oFeedOverride := 85;
           25:
               #oFeedOverride := 90;
           27:
               #oFeedOverride := 95;
           26:
               #oFeedOverride := 100;
           30:
               #oFeedOverride := 105;
           31:
               #oFeedOverride := 110;
           29:
               #oFeedOverride := 115;
           28:
               #oFeedOverride := 120;
       END_CASE;
   END_REGION
END_FUNCTION_BLOCK

FUNCTION_BLOCK "FB_LightsManagement"   // FB500, SCL
{ S7_Optimized_Access := 'TRUE' }
// stored: AutoNumber false, MemoryReserve 100, SetENOAutomatically false
BEGIN
   REGION Light Tower : Green light
       "DB_DigitalOutputs".sLightTowerGreen.sSWStatus :=
       "LBP_Chan1".E_ProgRunning
       OR "LBP_Chan1".E_ProgWait
       OR "LBP_Chan1".E_ProgStop
       OR "DB_McpKeyboardSignals".sLightTest.sKeySWStatus;
   END_REGION

   REGION Light Tower : Orange light
       "DB_DigitalOutputs".sLightTowerOrange.sSWStatus := ("DB_DataFromSafety".iEmergencyStopPowerLaser
       AND "DB_DataFromSafety".ShutterOpened
       AND "Clock_2.5Hz")
       OR "DB_McpKeyboardSignals".sLightTest.sKeySWStatus;
   END_REGION

   REGION Light Tower : Blue light
       "DB_DigitalOutputs".sLightTowerBlue.sSWStatus :=
       ("LBP_ModeGroup".E_AUTO
       AND ("LBP_Chan1".E_ProgRunning OR "LBP_Chan1".E_ProgWait)
       AND NOT "DB_DataFromSafety".EmergencyStop    
       AND "Clock_1Hz")
       OR "DB_McpKeyboardSignals".sLightTest.sKeySWStatus;
   END_REGION

   REGION Light Tower : White light
       "DB_DigitalOutputs".sLightTowerWhite.sSWStatus :=
       ("DB_PowerOn".sMachinePower
       AND "Clock_0.625Hz")
       OR "DB_McpKeyboardSignals".sLightTest.sKeySWStatus;
   END_REGION

   REGION Test LED light
       "DB_McpKeyboardSignals".sLightTest.sLedSWStatus := "DB_McpKeyboardSignals".sLightTest.sKeySWStatus;
   END_REGION

   REGION Machine lights (Key K15)
       IF "DB_McpKeyboardSignals".sK15_MachineLight.sKeySWTogglePositiveFront
           OR "DB_HmiKeyboardSignals".sK15_MachineLight.sKeySWTogglePositiveFront THEN
           "DB_DigitalOutputs".sMachineLight.sSWStatus := TRUE;
           "DB_DigitalOutputs".sMachineLightBack.sSWStatus := TRUE;
           "DB_McpKeyboardSignals".sK15_MachineLight.sKeySWToggleStatus := TRUE;
           "DB_HmiKeyboardSignals".sK15_MachineLight.sKeySWToggleStatus := TRUE;
       ELSIF "DB_McpKeyboardSignals".sK15_MachineLight.sKeySWToggleNegativeFront
           OR "DB_HmiKeyboardSignals".sK15_MachineLight.sKeySWToggleNegativeFront THEN
           "DB_DigitalOutputs".sMachineLight.sSWStatus := FALSE;
           "DB_DigitalOutputs".sMachineLightBack.sSWStatus := FALSE;
           "DB_McpKeyboardSignals".sK15_MachineLight.sKeySWToggleStatus := FALSE;
           "DB_HmiKeyboardSignals".sK15_MachineLight.sKeySWToggleStatus := FALSE;
       END_IF;
           "DB_McpKeyboardSignals".sK15_MachineLight.sLedSWStatus := "DB_DigitalOutputs".sMachineLight.sSWStatus;
           "DB_HmiKeyboardSignals".sK15_MachineLight.sLedSWStatus := "DB_DigitalOutputs".sMachineLight.sSWStatus;
   END_REGION

   REGION Camera lights (Key K12)    
       IF "LBP_Chan1".MDyn[50] THEN
           "DB_McpKeyboardSignals".sK12_ObservationCamera.sKeySWToggleStatus := TRUE;
           "DB_HmiKeyboardSignals".sK12b_ObservationCamera.sKeySWToggleStatus := TRUE;
       ELSIF "LBP_Chan1".MDyn[51] THEN
           "DB_McpKeyboardSignals".sK12_ObservationCamera.sKeySWToggleStatus := FALSE;
           "DB_HmiKeyboardSignals".sK12b_ObservationCamera.sKeySWToggleStatus := FALSE;
       END_IF;

       IF "DB_McpKeyboardSignals".sK12_ObservationCamera.sKeySWTogglePositiveFront
           OR "DB_HmiKeyboardSignals".sK12a_Backlight.sKeySWTogglePositiveFront THEN
           "DB_DigitalOutputs".sBacklight.sSWStatus := TRUE;
       ELSIF "DB_McpKeyboardSignals".sK12_ObservationCamera.sKeySWToggleNegativeFront
           OR "DB_HmiKeyboardSignals".sK12a_Backlight.sKeySWToggleNegativeFront THEN
           "DB_DigitalOutputs".sBacklight.sSWStatus := FALSE;
       END_IF;

       "DB_McpKeyboardSignals".sK12_ObservationCamera.sLedSWStatus := "DB_DigitalOutputs".sBacklight.sSWStatus;
       "DB_HmiKeyboardSignals".sK12a_Backlight.sLedSWStatus := "DB_DigitalOutputs".sBacklight.sSWStatus;

       IF "DB_McpKeyboardSignals".sK12_ObservationCamera.sKeySWTogglePositiveFront
           OR "DB_HmiKeyboardSignals".sK12b_ObservationCamera.sKeySWTogglePositiveFront THEN
           "DB_DigitalOutputs".sObservationCameraLight.sSWStatus := TRUE;
       ELSIF "DB_McpKeyboardSignals".sK12_ObservationCamera.sKeySWToggleNegativeFront
           OR "DB_HmiKeyboardSignals".sK12b_ObservationCamera.sKeySWToggleNegativeFront THEN
           "DB_DigitalOutputs".sObservationCameraLight.sSWStatus := FALSE;
       END_IF;

       "DB_McpKeyboardSignals".sK12_ObservationCamera.sLedSWStatus := "DB_DigitalOutputs".sObservationCameraLight.sSWStatus;
       "DB_HmiKeyboardSignals".sK12b_ObservationCamera.sLedSWStatus := "DB_DigitalOutputs".sObservationCameraLight.sSWStatus;
   END_REGION

   REGION Ack blue button AND red light tower blinking
       "DB_McpKeyboardSignals".sAlarmReset.sLedSWStatus :=
           (( "DB_Alarms".sAlarmsLevel1
           OR "DB_Alarms".sAlarmsLevel2
           OR "DB_Alarms".sAlarmsLevel3
           OR "DB_Alarms".sAlarmsLevel4
           OR "DB_Alarms".sAlarmsLevel5
           OR "DB_Alarms".sAlarmsLevel6)
           AND "Clock_1Hz")
           OR "DB_McpKeyboardSignals".sLightTest.sKeySWStatus;

           "DB_DigitalOutputs".sLightTowerRed.sSWStatus :=
           (( "DB_Alarms".sAlarmsLevel2
           OR "DB_Alarms".sAlarmsLevel3
           OR "DB_Alarms".sAlarmsLevel4
           OR "DB_Alarms".sAlarmsLevel5
           OR "DB_Alarms".sAlarmsLevel6)
           AND "Clock_1Hz")
           OR "DB_McpKeyboardSignals".sLightTest.sKeySWStatus;
   END_REGION
END_FUNCTION_BLOCK

FUNCTION_BLOCK "FB_MainDoorManagement"   // FB510, SCL
{ S7_Optimized_Access := 'TRUE' }
// stored: AutoNumber false, MemoryReserve 100, SetENOAutomatically false
   VAR
      FT_AxisDesactivated { S7_SetPoint := 'True'} : F_TRIG;
      sDoorNotLocked : Bool;
      sLockAutoFrontDoor : Bool;
   END_VAR
BEGIN
   REGION Key[13] Management
       // Key disabled
       "DB_McpKeyboardSignals".sK13_MainDoor.sKeyDisable := NOT "LBP_ModeGroup".E_JOG OR "DB_GestionWorkingModes".sMCP_KxxKeysDisable;

       // Set Door unlock when axis are desactivated
    //   #FTAxisDesactivated(CLK :="DB_DigitalOutputs".Axis_Activation.SWStatus,       WFA A revoir
     //                      Q => "DB_McpKeyboardSignals".K13_MainDoor.KeySWToggleStatus);
   END_REGION

   REGION Unlock / Lock Front Door
       IF "DB_McpKeyboardSignals".sK13_MainDoor.sKeySWTogglePositiveFront
           OR NOT "DB_DataFromSafety".EmergencyStop
           OR "DB_HMISetting".UnlockDoorReq
      //     OR NOT "DB_DigitalOutputs".Axis_Activation.SWStatus       WFA A rajouter 
           OR NOT "DB_DigitalInputs".sFrontDoorClosed.sSWStatus THEN
           "DB_DataToSafety".FrontDoorLock := FALSE;
       ELSIF "DB_McpKeyboardSignals".sK13_MainDoor.sKeySWToggleNegativeFront
           OR #sLockAutoFrontDoor
           OR "DB_HMISetting".LockDoorReq
           AND "DB_DataFromSafety".iFrontDoorClosed
           AND "DB_DigitalInputs".sFrontDoorClosed.sSWStatus THEN
           "DB_DataToSafety".FrontDoorLock := TRUE;
       END_IF;
       "DB_HMISetting".UnlockDoorReq := FALSE;
       "DB_HMISetting".LockDoorReq := FALSE;
   END_REGION

   REGION Led[13] Management
           // OFF : Door Closed and Locked
           // Blink : Door Closed and not Locked
           // ON : Door Open
       "DB_McpKeyboardSignals".sK13_MainDoor.sLedSWStatus :=
       NOT "DB_DataToSafety".FrontDoorLock
       AND ("DB_DataFromSafety".iFrontDoorClosed AND "Clock_1Hz")
       OR NOT "DB_DataFromSafety".iFrontDoorClosed;
   END_REGION

   REGION Alarm messages
       IF NOT "LBP_ModeGroup".E_AUTO THEN
           "LBP_AlarmMsgs".UserA[0].A70UUxx[61] := FALSE;  // Msg: 700061 "Door not locked, cycle start automatically locks main door"
           "LBP_AlarmMsgs".UserA[0].A70UUxx[62] := FALSE;  // Msg: 700062 "Automatic locking of main door on start cycle"
           "LBP_AlarmMsgs".UserA[0].A70UUxx[63] := FALSE;  // Msg: 700063 "Main door open, start cycle not allowed, please close the main door"
       END_IF;

       // Msg: "700061 - Door not locked, cycle start automatically locks main door" 
       "LBP_AlarmMsgs".UserA[0].A70UUxx[61] :=
       NOT "DB_DigitalInputs".sFrontDoorLocked.sSWStatus
       AND "DB_DigitalInputs".sFrontDoorClosed.sSWStatus;

       // Front Door Not Locked
       IF ("DB_DigitalInputs".sFrontDoorLocked.sSWStatus AND #sDoorNotLocked AND "LBP_Chan1".E_ProgRunning)
           OR "MCP1_In".reset THEN
           #sDoorNotLocked := FALSE;
       ELSIF NOT "DB_DigitalInputs".sFrontDoorLocked.sSWStatus AND "DB_DigitalInputs".sFrontDoorClosed.sSWStatus AND "MCP1_In".cycleStart THEN
           #sDoorNotLocked := TRUE;
       END_IF;

       // Msg: 700062 "Automatic locking of main door on start cycle"
       "LBP_AlarmMsgs".UserA[0].A70UUxx[62] := NOT "DB_DigitalInputs".sFrontDoorLocked.sSWStatus AND "DB_DigitalInputs".sFrontDoorClosed.sSWStatus AND ("MCP1_In".cycleStart OR "DB_McpKeyboardSignals".sStartCycle.sKeySWStatus);
       #sLockAutoFrontDoor := "LBP_AlarmMsgs".UserA[0].A70UUxx[62];

       // Msg: 700063 "Main door open, start cycle not allowed, please close the main door"
       IF NOT "DB_DigitalInputs".sFrontDoorLocked.sSWStatus AND NOT "DB_DigitalInputs".sFrontDoorClosed.sSWStatus AND ("MCP1_In".cycleStart OR "DB_McpKeyboardSignals".sStartCycle.sKeySWStatus) THEN
           "LBP_AlarmMsgs".UserA[0].A70UUxx[63] := TRUE;
       ELSIF "DB_DigitalInputs".sFrontDoorClosed.sSWStatus THEN
           "LBP_AlarmMsgs".UserA[0].A70UUxx[63] := FALSE;
       END_IF;
   END_REGION
END_FUNCTION_BLOCK

FUNCTION_BLOCK "FB_Tracability"   // FB700, SCL
{ S7_Optimized_Access := 'TRUE' }
// stored: AutoNumber false, MemoryReserve 100, SetENOAutomatically false
   VAR_INPUT
      iCondTransfertExtInTo1 : Bool;
      iCondTransfertExtInTo2 : Bool;
      iCondTransfert1To3 : Bool;
      iCondTransfert2To3 : Bool;
      iCondTransfert3To4 : Bool;
      iCondTransfert4To5 : Bool;
      iCondTransfert5To6 : Bool;
      iCondTransfert5To7 : Bool;
      iCondTransfert6ToExtOut : Bool;
      iCondTransfert7ToExtOut : Bool;
   END_VAR
   VAR
      sRT_ConditionExtInTo1 : R_TRIG;
      sRT_ConditionExtInTo2 { S7_SetPoint := 'True'} : R_TRIG;
      sRT_Condition1To3 { S7_SetPoint := 'True'} : R_TRIG;
      sRT_Condition2To3 { S7_SetPoint := 'True'} : R_TRIG;
      sRT_Condition3To4 { S7_SetPoint := 'True'} : R_TRIG;
      sRT_Condition4To5 { S7_SetPoint := 'True'} : R_TRIG;
      sRT_Condition5To6 { S7_SetPoint := 'True'} : R_TRIG;
      sRT_Condition5To7 { S7_SetPoint := 'True'} : R_TRIG;
      sRT_Condition6ToExtOut { S7_SetPoint := 'True'} : R_TRIG;
      sRT_Condition7ToExtOut { S7_SetPoint := 'True'} : R_TRIG;
      sIndex : Int;
      sCheckTransfertExtInTo1 : Bool;
      sCheckTransfertExtInTo2 : Bool;
      sCheckTransfert1To3 : Bool;
      sCheckTransfert2To3 : Bool;
      sCheckTransfert3To4 : Bool;
      sCheckTransfert4To5 : Bool;
      sCheckTransfert5To6 : Bool;
      sCheckTransfert5To7 : Bool;
      sCheckTransfert6ToExtOut : Bool;
      sCheckTransfert7ToExtOut : Bool;
      sLaserTime : "FB_TimeCounter";
      sMemoPartDMC { S7_SetPoint := 'True'} : Array[0..19] of Byte;
   END_VAR
   VAR RETAIN
      sIEC_CounterCycleLaser { S7_SetPoint := 'True'} : TONR_TIME;
      sIEC_CounterCycleTime { S7_SetPoint := 'True'} : TONR_TIME;
      sStartCounterCycleLaser { S7_SetPoint := 'True'} : Bool;
      sStartCounterCycleTime { S7_SetPoint := 'True'} : Bool;
   END_VAR
   VAR_TEMP
      tFailCodePart : Int;
      tFailCodeBackwall : Int;
      tHoleNumber : Int;
      tMeasureZ : Real;
      tWOZ : Int;
      tWOC : Int;
      tTotalCycleTimeCh1 : Int;
      tLaserCycleTimeCh1 : Int;
   END_VAR
   VAR CONSTANT
      POSITION_NUMBER : Int := 7;
   END_VAR
BEGIN
   REGION Reset data Postions station 1
       // Positions :
           //  1 : Shuttle 1 Undrilled Part
           //  2 : Shuttle 2 Undrilled Part
           //  3 : Gripper   Undrilled Part
           //  4 : Fixture
           //  5 : Gripper   Drilled Part
           //  6 : Shuttle 1 Drilled Part
           //  7 : Shuttle 2 Drilled Part

       IF "LBP_Chan1".A_Ref THEN
           #sCheckTransfertExtInTo1 := FALSE;     
           #sCheckTransfertExtInTo2 := FALSE;     
           #sCheckTransfert1To3 := FALSE;            
           #sCheckTransfert2To3 := FALSE;           
           #sCheckTransfert3To4 := FALSE;           
           #sCheckTransfert4To5 := FALSE;            
           #sCheckTransfert5To6 := FALSE;        
           #sCheckTransfert5To7 := FALSE;         
           #sCheckTransfert6ToExtOut := FALSE;   
           #sCheckTransfert7ToExtOut := FALSE;     
           FOR #sIndex := 0 TO #POSITION_NUMBER DO
               "FC_ResetPositionData"(iDataPosition := #sIndex);
           END_FOR;
       END_IF;
   END_REGION

   REGION Transfert Postions data station 1 
       IF #sCheckTransfert1To3 THEN
           // Transfert data from position 1 To 3 - Shuttle 1 to Loading Gripper 
           "DB_DataPositions".Position[3] := "DB_DataPositions".Position[1];
           // Reset data in position 1
           "FC_ResetPositionData"(iDataPosition := 1);
           #sCheckTransfert1To3 := FALSE;
       END_IF;

       IF #sCheckTransfert2To3 THEN
           // Transfert data from position 2 To 3 - Shuttle 2 to Loading Gripper 
           "DB_DataPositions".Position[3] := "DB_DataPositions".Position[2];
           // Reset data in position 2
           "FC_ResetPositionData"(iDataPosition := 2);
           #sCheckTransfert2To3 := FALSE;
       END_IF;

       IF #sCheckTransfert3To4 THEN
           // Transfert data from position 3 To 4 - Loading Gripper to Fixture
           "DB_DataPositions".Position[4] := "DB_DataPositions".Position[3];
           // Reset data in position 3
           "FC_ResetPositionData"(iDataPosition := 3);
           #sCheckTransfert3To4 := FALSE;
       END_IF;

       IF #sCheckTransfert4To5 THEN
           // Transfert data from position 4 To 5 - Fixture to Unloading Gripper
           "DB_DataPositions".Position[5] := "DB_DataPositions".Position[4];
           // Reset data in position 4
           "FC_ResetPositionData"(iDataPosition := 4);
           #sCheckTransfert4To5 := FALSE;
       END_IF;

       IF #sCheckTransfert5To6 THEN
           // Transfert data from position 5 To 6 - Unloading Gripper to Shuttle 1
           "DB_DataPositions".Position[6] := "DB_DataPositions".Position[5];
           // Reset data in position 5
           "FC_ResetPositionData"(iDataPosition := 5);
           #sCheckTransfert5To6 := FALSE;
       END_IF;

       IF #sCheckTransfert5To7 THEN
           // Transfert data from position 5 To 7 - Unloading Gripper to Shuttle 2
           "DB_DataPositions".Position[7] := "DB_DataPositions".Position[5];
           // Reset data in position 5
           "FC_ResetPositionData"(iDataPosition := 5);
           #sCheckTransfert5To7 := FALSE;
       END_IF;

       IF #sCheckTransfert6ToExtOut THEN
           // Shift of the the array for the new final part
           FOR #sIndex := 98 TO 0 BY -1 DO
               "DB_DataFinalPart".FinalPart[#sIndex + 1] := "DB_DataFinalPart".FinalPart[#sIndex];
           END_FOR;
           // Transfert data from position 6 TO the DB final part - Shuttle 1 to DB final part
           "DB_DataFinalPart".FinalPart[0] := "DB_DataPositions".Position[6];
           "FC_ResetPositionData"(iDataPosition := 6);
           #sCheckTransfert6ToExtOut := FALSE;
       END_IF;

       IF #sCheckTransfert7ToExtOut THEN
           // Shift of the the array for the new final part
           FOR #sIndex := 98 TO 0 BY -1 DO
               "DB_DataFinalPart".FinalPart[#sIndex + 1] := "DB_DataFinalPart".FinalPart[#sIndex];
           END_FOR;
           // Transfert data from position 7 TO the DB final part - Shuttle 2 to DB final part
           "DB_DataFinalPart".FinalPart[0] := "DB_DataPositions".Position[7];
           "FC_ResetPositionData"(iDataPosition := 7);
           #sCheckTransfert7ToExtOut := FALSE;
       END_IF;
   END_REGION

   REGION Condition for the Transfert Postions data
       // Conditions from Ext To position 1 - External Loader to Shuttle 1
       #sRT_ConditionExtInTo1(CLK := #iCondTransfertExtInTo1);
       IF #sRT_ConditionExtInTo1.Q THEN
           #sCheckTransfertExtInTo1 := TRUE;
       END_IF;

       // Conditions from Ext To position 2 - External Loader to Shuttle 2
       #sRT_ConditionExtInTo2(CLK := #iCondTransfertExtInTo2);
       IF #sRT_ConditionExtInTo2.Q THEN
           #sCheckTransfertExtInTo2 := TRUE;
       END_IF;

       // Conditions from position 1 To 3 - Shuttle 1 to Loading Gripper 
       #sRT_Condition1To3(CLK:=#iCondTransfert1To3);
       IF #sRT_Condition1To3.Q THEN
           #sCheckTransfert1To3 := TRUE;
       END_IF;

       // Conditions from position 2 To 3 - Shuttle 2 to Loading Gripper 
       #sRT_Condition2To3(CLK := #iCondTransfert2To3);
       IF #sRT_Condition2To3.Q THEN
           #sCheckTransfert2To3 := TRUE;
       END_IF;

       // Conditions from position 3 To 4 - Loading Gripper to Fixture
       #sRT_Condition3To4(CLK := #iCondTransfert3To4);
       IF #sRT_Condition3To4.Q THEN
           #sCheckTransfert3To4 := TRUE;
       END_IF;

       // Conditions from position 4 To 5 - Fixture to Unloading Gripper
       #sRT_Condition4To5(CLK := #iCondTransfert4To5);
       IF #sRT_Condition4To5.Q THEN
           #sCheckTransfert4To5 := TRUE;
       END_IF;

       // Conditions from position 5 To 6 - Unloading Gripper to Shuttle 1
       #sRT_Condition5To6(CLK := #iCondTransfert5To6);
       IF #sRT_Condition5To6.Q THEN
           #sCheckTransfert5To6 := TRUE;
       END_IF;

       // Conditions from position 5 To 7 - Unloading Gripper to Shuttle 2
       #sRT_Condition5To7(CLK := #iCondTransfert5To7);
       IF #sRT_Condition5To7.Q THEN
           #sCheckTransfert5To7 := TRUE;
       END_IF;

       // Conditions from position 6 To Ext - Shuttle 1 to External Loader
       #sRT_Condition6ToExtOut(CLK := #iCondTransfert6ToExtOut);
       IF #sRT_Condition6ToExtOut.Q THEN
           #sCheckTransfert6ToExtOut := TRUE;
       END_IF;

       // Conditions from position 7 To Ext - Shuttle 2 to External Loader
       #sRT_Condition7ToExtOut(CLK := #iCondTransfert7ToExtOut);
       IF #sRT_Condition7ToExtOut.Q THEN
           #sCheckTransfert7ToExtOut := TRUE;
       END_IF;
   END_REGION

   REGION Update Data
       // Détection nouvelle pièce
       IF #sCheckTransfertExtInTo1 THEN
           // Initialisation de la donnée de la pièce sur shuttle 1
           "DB_DataPositions".Position[1].DMC := "DB_SonplasMain".sSonplasLoader.iPartInDMC_CodeShuttle1;
           #sCheckTransfertExtInTo1 := FALSE;
       END_IF;
       IF #sCheckTransfertExtInTo2 THEN
           // Initialisation de la donnée de la pièce sur shuttle 2
           "DB_DataPositions".Position[2].DMC := "DB_SonplasMain".sSonplasLoader.iPartInDMC_CodeShuttle2;
           #sCheckTransfertExtInTo2 := FALSE;
       END_IF;
       // Fail code part
       IF "LBP_Chan1".MDyn[69] THEN
           #tFailCodePart := REAL_TO_INT("LBP_Chan1".H1);
       END_IF;
       // Measure Z
       IF "LBP_Chan1".MDyn[98] THEN
           #tHoleNumber := REAL_TO_INT("LBP_Chan1".H1);
           #tMeasureZ := "LBP_Chan1".H2;
       END_IF;
       // WOZ
       IF "LBP_Chan1".MDyn[37] THEN
           #tWOZ := REAL_TO_INT("LBP_Chan1".H1);
       END_IF;
       // WOC
       IF "LBP_Chan1".MDyn[38] THEN
           #tWOC := REAL_TO_INT("LBP_Chan1".H1);
       END_IF;
       "DB_DataPositions".Position[4].FailCode := #tFailCodePart;
       "DB_DataPositions".Position[4].WOZ_Measure := #tWOZ;
       "DB_DataPositions".Position[4].WOC_Measure := #tWOC;
       #sMemoPartDMC:= "DB_DataPositions".Position[4].DMC;
       // Counter if cycle time
       IF "LBP_Chan1".MDyn[72] THEN             // M72 : Start counter of cycle time
           #sStartCounterCycleTime := TRUE;
       ELSIF "LBP_Chan1".MDyn[73] THEN          // M73 : Stop counter of cycle time
           #sStartCounterCycleTime := FALSE;
       END_IF;
       #sIEC_CounterCycleTime(IN:=#sStartCounterCycleTime,
                              R:=NOT #sStartCounterCycleTime,
                              PT:=t#10m);
       // Counter of cycle laser
       IF "LBP_Chan1".MDyn[71] THEN            // M71 : Start calculation laser time 
           #sStartCounterCycleLaser := TRUE;
       ELSIF "LBP_Chan1".MDyn[68] THEN         // M68 : Set Lasered (Tracability)
           #sStartCounterCycleLaser := FALSE;
       END_IF;
       #sIEC_CounterCycleLaser(IN:=#sStartCounterCycleLaser,
                               R:=NOT #sStartCounterCycleLaser,
                               PT:=t#10m);
       // Mesure ZED Backwall PAS UTILISE SUR FL0153 A SUPPRIMER
       IF "LBP_Chan1".MDyn[29] THEN
           #tFailCodeBackwall := REAL_TO_INT("LBP_Chan1".H1);
       END_IF;
       // Close unload gripper
       IF "DB_DataPositions".Position[4].DMC = #sMemoPartDMC THEN
           IF "LBP_Chan1".MDyn[82] THEN
               "DB_DataPositions".Position[4].TotalCycleTime := TIME_TO_INT(#sIEC_CounterCycleTime.ET);
               "DB_DataPositions".Position[4].LaserCycleTime := TIME_TO_INT(#sIEC_CounterCycleLaser.ET);
           END_IF;
           "DB_DataPositions".Position[4].FailCodeBackwall := #tFailCodeBackwall;

       ELSIF "DB_DataPositions".Position[5].DMC = #sMemoPartDMC THEN
           IF "LBP_Chan1".MDyn[82] THEN
               "DB_DataPositions".Position[5].TotalCycleTime := TIME_TO_INT(#sIEC_CounterCycleTime.ET);
               "DB_DataPositions".Position[5].LaserCycleTime := TIME_TO_INT(#sIEC_CounterCycleLaser.ET);
           END_IF;
           "DB_DataPositions".Position[5].FailCodeBackwall := #tFailCodeBackwall;
       END_IF;
   END_REGION
END_FUNCTION_BLOCK

FUNCTION_BLOCK "FB_SonplasMain"   // FB42, SCL
{ S7_Optimized_Access := 'TRUE' }
// stored: MemoryReserve 100, SetENOAutomatically false
   VAR
      sSonplasLoader : "FB_SonplasLoader";
      iDMC_CodeShuttle1 { S7_SetPoint := 'True'} : String;
      iDMC_CodeShuttle2 : String;
      iDMC_Code : String;
      oDMC_CodeShuttle1 : String;
      oDMC_CodeShuttle2 : String;
      oDMC_Code : String;
   END_VAR
   VAR_TEMP
      tRetMov : Int;
      tIndex : Int;
   END_VAR
BEGIN
   REGION Description head
       //==================================================================================
       // POSALUX Swiss SA / (C) Copyright 2025
       //----------------------------------------------------------------------------------
       // Title: Digital Inputs mapping
       // Comment/Function: Digital Inputs mapping
       // Author: Fabien WALDT
       // Engineering: TIA Portal v17
       //----------------------------------------------------------------------------------
       // Change log table:
       // Version  | Date     | Expert in charge | Changes applied
       // ---------|----------|------------------|-----------------------------------------
       // 00.00.01 | 20250423 | WFA              | First released version
       // =================================================================================
   END_REGION

   REGION DMC Reading
      // Transfer DMC Code Shuttle 1 (IB204-IB223)
       // #tRetMov := MOVE_BLK_VARIANT(SRC := P# I204.0 BYTE 20, // WAF COMENTAIRE POUR TESTS TRACABILITE
       //                              COUNT := 20,
       //                              SRC_INDEX := 0,
       //                              DEST_INDEX := 0,
       //                              DEST => #sSonplasLoader.iPartInDMC_CodeShuttle1);

       // String Conversion
       #iDMC_CodeShuttle1 := '';
       FOR #tIndex := 0 TO 19 DO
           IF #sSonplasLoader.iPartInDMC_CodeShuttle1[#tIndex] <> 0 THEN
               #iDMC_CodeShuttle1 := CONCAT(IN1 := #iDMC_CodeShuttle1, IN2 := CHAR_TO_STRING(BYTE_TO_CHAR(#sSonplasLoader.iPartInDMC_CodeShuttle1[#tIndex])));
           END_IF;
       END_FOR;

      // Transfer DMC Code Shuttle 2 (IB224-IB243)
       // #tRetMov := MOVE_BLK_VARIANT(SRC := P# I224.0 BYTE 20, // WAF COMENTAIRE POUR TESTS TRACABILITE
       //                             COUNT := 20,
       //                             SRC_INDEX := 0,
       //                             DEST_INDEX := 0,
       //                             DEST => #sSonplasLoader.iPartInDMC_CodeShuttle2);


       // String Conversion
      #iDMC_CodeShuttle2 := '';
       FOR #tIndex := 0 TO 19 DO
           IF #sSonplasLoader.iPartInDMC_CodeShuttle2[#tIndex] <> 0 THEN
               #iDMC_CodeShuttle2 := CONCAT(IN1 := #iDMC_CodeShuttle2, IN2 := CHAR_TO_STRING(BYTE_TO_CHAR(#sSonplasLoader.iPartInDMC_CodeShuttle2[#tIndex])));
           END_IF;
       END_FOR;

       // Transfer DMC Code (IB247-IB266)
       #tRetMov := MOVE_BLK_VARIANT(SRC := P# I247.0 BYTE 20,
                                    COUNT := 20,
                                    SRC_INDEX := 0,
                                    DEST_INDEX := 0,
                                    DEST => #sSonplasLoader."iPartInDMC Code");


       // String Conversion
       #iDMC_Code := '';
       FOR #tIndex := 0 TO 19 DO
           IF #sSonplasLoader."iPartInDMC Code"[#tIndex] <> 0 THEN
               #iDMC_Code := CONCAT(IN1 := #iDMC_Code, IN2 := CHAR_TO_STRING(BYTE_TO_CHAR(#sSonplasLoader."iPartInDMC Code"[#tIndex])));
           END_IF;
       END_FOR;

   END_REGION

   REGION Sonplas Loader
       #sSonplasLoader(iOperateInDiagDPCoupler:="DB_DigitalInputsSonplas".sSonplasDiagDPCoupler.sSWStatus,
                       iOperateInReady:="DB_DigitalInputsSonplas".sSonplasReady.sSWStatus,
                       iOperateInNoEStop:="DB_DigitalInputsSonplas".sSonplasNoEStop.sSWStatus,
                       iOperateInDoorsClosed:="DB_DigitalInputsSonplas".sSonplasDoorsClosed.sSWStatus,
                       iOperateInRunError:="DB_DigitalInputsSonplas".sSonplasRunError.sSWStatus,
                       iOperateInOutCollision:="DB_DigitalInputsSonplas".sSonplasOutCollision.sSWStatus OR "DB_WAF".Sonplas.OperateInOutCollision,
                       iPartInShuttle1Finished:="DB_DigitalInputsSonplas".sSonplasShuttle1Finished.sSWStatus,
                       iPartInShuttle2Finished:="DB_DigitalInputsSonplas".sSonplasShuttle2Finished.sSWStatus,
                       iMeasureInFlowResultAvail:="DB_DigitalInputsSonplas".sSonplasFlowResultAvail.sSWStatus,
                       iMeasureInFlowResult:= WORD_TO_INT(SWAP_WORD("AI_SonplasFlowResult")),
                       oOperateOutDiagDPCoupler=>"DB_DigitalOutputs".sSonplasDiagDPCoupler.sSWStatus,
                       oOperateOutReady=>"DB_DigitalOutputs".sSonplasReady.sSWStatus,
                       oOperateOutNoEStop=>"DB_DigitalOutputs".sSonplasNoEStop.sSWStatus,
                       oOperateOutDoorsClosed=>"DB_DigitalOutputs".sSonplasDoorsClosed.sSWStatus,
                       oOperateOutRunError=>"DB_DigitalOutputs".sSonplasRunError.sSWStatus,
                       oPartOutShuttle1InPos=>"DB_DigitalOutputs".sSonplasShuttle1InPos.sSWStatus,
                       oPartOutPart1OK=>"DB_DigitalOutputs".sSonplasPart1OK.sSWStatus,
                       oPartOutPart1NOK=>"DB_DigitalOutputs".sSonplasPart1NOK.sSWStatus,
                       oPartOutShuttle2InPos=>"DB_DigitalOutputs".sSonplasShuttle2InPos.sSWStatus,
                       oPartOutPart2OK=>"DB_DigitalOutputs".sSonplasPart2OK.sSWStatus,
                       oPartOutPart2NOK=>"DB_DigitalOutputs".sSonplasPart2NOK.sSWStatus,
                       oMeasureOutResultAccepted=>"DB_DigitalOutputsSonplas".Sonplas_ResultAccepted.sSWStatus);
   END_REGION

   REGION DMC Writing   
       // Transfer DMC Code Shuttle 1 (QB204-QB223)
       FOR #tIndex := 1 TO LEN(#oDMC_CodeShuttle1) DO
           #sSonplasLoader.oPartOutDMC_CodeShuttle1[#tIndex - 1] := CHAR_TO_BYTE(#oDMC_CodeShuttle1[#tIndex]);
       END_FOR;

       #tRetMov := MOVE_BLK_VARIANT(SRC := #sSonplasLoader.oPartOutDMC_CodeShuttle1,
                                    COUNT := 20,
                                    SRC_INDEX := 0,
                                    DEST_INDEX := 0,
                                    DEST => P# Q204.0 BYTE 20);

   // Transfer DMC Code Shuttle 2 (QB224-QB243)
   FOR #tIndex := 1 TO LEN(#oDMC_CodeShuttle2) DO
       #sSonplasLoader.oPartOutDMC_CodeShuttle2[#tIndex - 1] := CHAR_TO_BYTE(#oDMC_CodeShuttle2[#tIndex]);
   END_FOR;

   #tRetMov := MOVE_BLK_VARIANT(SRC := #sSonplasLoader.oPartOutDMC_CodeShuttle2,
                                COUNT := 20,
                                SRC_INDEX := 0,
                                DEST_INDEX := 0,
                                DEST => P# Q224.0 BYTE 20);

   // Transfer DMC Code (QB247-QB266)
   FOR #tIndex := 1 TO LEN(#oDMC_Code) DO
       #sSonplasLoader.oPartOutDMC_Code[#tIndex - 1] := CHAR_TO_BYTE(#oDMC_Code[#tIndex]);
   END_FOR;

   #tRetMov := MOVE_BLK_VARIANT(SRC := #sSonplasLoader.oPartOutDMC_Code,
                                COUNT := 20,
                                SRC_INDEX := 0,
                                DEST_INDEX := 0,
                                DEST => P# Q247.0 BYTE 20);
   END_REGION
END_FUNCTION_BLOCK

FUNCTION_BLOCK "FB_SonplasLoader"   // FB36, SCL
{ S7_Optimized_Access := 'TRUE' }
// stored: MemoryReserve 100, SetENOAutomatically false
   VAR_INPUT
      iOperateInDiagDPCoupler : Bool;
      iOperateInReady : Bool;
      iOperateInNoEStop : Bool;
      iOperateInDoorsClosed : Bool;
      iOperateInRunError : Bool;
      iOperateInOutCollision : Bool;
      iPartInShuttle1Finished : Bool;
      iPartInShuttle2Finished : Bool;
      iPartInDMC_CodeShuttle1 : Array[0..19] of Byte;
      iPartInDMC_CodeShuttle2 : Array[0..19] of Byte;
      "iPartInDMC Code" : Array[0..19] of Byte;
      iMeasureInFlowResultAvail : Bool;
      iMeasureInFlowResult : Int;
      iMeasureInDMC_Code : Array[0..19] of Byte;
   END_VAR
   VAR_OUTPUT
      oOperateOutDiagDPCoupler : Bool;
      oOperateOutReady : Bool;
      oOperateOutNoEStop : Bool;
      oOperateOutDoorsClosed : Bool;
      oOperateOutRunError : Bool;
      oPartOutShuttle1InPos : Bool;
      oPartOutPart1OK : Bool;
      oPartOutPart1NOK : Bool;
      oPartOutShuttle2InPos : Bool;
      oPartOutPart2OK : Bool;
      oPartOutPart2NOK : Bool;
      oPartOutDMC_CodeShuttle1 : Array[0..19] of Byte;
      oPartOutDMC_CodeShuttle2 : Array[0..19] of Byte;
      oPartOutDMC_Code : Array[0..19] of Byte;
      oMeasureOutResultAccepted : Bool;
   END_VAR
   VAR
      sAutomaticMode : Bool;
      sSemiAutoMode : Bool;
      sLastFlowValue : Int;
      sRT_MeasureInFlowResultAvail : R_TRIG;
      sDiagDPCoupler : Bool;
      sReady : Bool;
      sNoEStop : Bool;
      sDoorsClosed : Bool;
      sRunError : Bool;
      sOutCollision : Bool;
      sShuttle1Finished : Bool;
      sShuttle2Finished : Bool;
      sFlowResultAvail : Bool;
      sFlowResult : Real;
      sMeasureDMC_Code : Array[0..19] of Byte;
   END_VAR
   VAR_TEMP
      tIndex : Int;
   END_VAR
BEGIN
   REGION Description header 
       //==================================================================================
       // POSALUX Swiss SA / (C) Copyright 2025
       //----------------------------------------------------------------------------------
       // Title: Initialization of axis
       // Comment/Function: FB_Ext_Loader
       // Author: Fabien WALDT
       // Engineering: TIA Portal v19
       //----------------------------------------------------------------------------------
       // Change log table:
       // Version  | Date     | Expert in charge | Changes applied
       // ---------|----------|------------------|-----------------------------------------
       // 00.00.01 | 20250917 | WFA              | First released version
       // =================================================================================
   END_REGION

   REGION Select automatic / semi automatic mode
       // Keys disabled WFA
       // IF ("LBP_Chan1".E_ProgWait
       //     OR "LBP_Chan1".E_ProgRunning
       //     OR "LBP_Chan1".E_ProgStop)
       //     AND "LBP_ModeGroup".E_AUTO THEN
       //     "DB_McpKeyboardSignals".K10_LoaderAuto.KeyDisable := TRUE;
       //     "DB_McpKeyboardSignals".K11_LoaderSemiAuto.KeyDisable := TRUE;
       //     "DB_HmiKeyboardSignals".K10_LoaderAuto.KeyDisable := TRUE;
       //     "DB_HmiKeyboardSignals".K11_LoaderSemiAuto.KeyDisable := TRUE;
       // ELSE
       //     "DB_McpKeyboardSignals".K10_LoaderAuto.KeyDisable := FALSE;
       //     "DB_McpKeyboardSignals".K11_LoaderSemiAuto.KeyDisable := FALSE;
       //     "DB_HmiKeyboardSignals".K10_LoaderAuto.KeyDisable := FALSE;
       //     "DB_HmiKeyboardSignals".K11_LoaderSemiAuto.KeyDisable := FALSE;
       // END_IF;

       // Mode selection
       #sAutomaticMode := "DB_McpKeyboardSignals".sK10_LoaderAuto.sKeySWToggleStatus;
       // OR "DB_OPC_Machine".State.Current.CurrrentLoadingMode = 1;

       #sSemiAutoMode := "DB_McpKeyboardSignals".sK11_LoaderSemiAuto.sKeySWToggleStatus;
       // OR "DB_OPC_Machine".State.Current.CurrrentLoadingMode = 2;

       // Flip-flop mode selection
       IF "DB_McpKeyboardSignals".sK10_LoaderAuto.sKeySWNegativeFront THEN
           "DB_McpKeyboardSignals".sK11_LoaderSemiAuto.sKeySWToggleStatus := FALSE;
       END_IF;
       IF "DB_McpKeyboardSignals".sK11_LoaderSemiAuto.sKeySWNegativeFront THEN
           "DB_McpKeyboardSignals".sK10_LoaderAuto.sKeySWToggleStatus := FALSE;
       END_IF;

       // LED Management
       "DB_McpKeyboardSignals".sK10_LoaderAuto.sLedSWStatus := "DB_WorkingModes".sAuto;
       "DB_McpKeyboardSignals".sK11_LoaderSemiAuto.sLedSWStatus := "DB_WorkingModes".sSemiAuto;

   END_REGION

   REGION Sonplas Inputs
       REGION Operating_Mode
           // Diagnostic bit DP / DP coupler
           #sDiagDPCoupler := #iOperateInDiagDPCoupler;

           // Sonplas ready
           #sReady := #iOperateInReady;

           // No emergency stop at Sonplas
           #sNoEStop := #iOperateInNoEStop;

           // Safety doors closed at Sonplas
           #sDoorsClosed := #iOperateInDoorsClosed;

           // Running error
           #sRunError := #iOperateInRunError;

           // Loader outside collision area
           #sOutCollision := #iOperateInOutCollision;
       END_REGION

       REGION Part Exchange
           // Posalux Shuttle 1 finished
           #sShuttle1Finished := #iPartInShuttle1Finished;

           // Posalux Shuttle 2 finished
           #sShuttle2Finished := #iPartInShuttle2Finished;
       END_REGION

       REGION Measure
           // Flow result available
           #sFlowResultAvail := #iMeasureInFlowResultAvail;

           // Flow Result
           #sFlowResult := INT_TO_REAL(#iMeasureInFlowResult);

           // Measure DMC Code
           #sMeasureDMC_Code := #iMeasureInDMC_Code;
       END_REGION
   END_REGION

   REGION Measure
       IF #sAutomaticMode OR "DB_WAF".BwLoader.Auto THEN
           #sRT_MeasureInFlowResultAvail(CLK := #sFlowResultAvail);
           IF #sRT_MeasureInFlowResultAvail.Q THEN
               FOR #tIndex := 0 TO 100 DO
                   IF "DB_DataFinalPart".FinalPart[#tIndex].DMC = #"iPartInDMC Code" THEN
                       "DB_DataFinalPart".FinalPart[#tIndex].FlowResult := #sFlowResult;
                       #oMeasureOutResultAccepted := TRUE;
                       EXIT;
                   // ELSE
                       // Product not found WFA A TRAITER
                   END_IF;
               END_FOR;
           ELSIF NOT #iMeasureInFlowResultAvail THEN
               #oMeasureOutResultAccepted := FALSE;
           END_IF;
       ELSE
           #oMeasureOutResultAccepted := FALSE;
       END_IF;
   END_REGION

   REGION Alarmes Messages
       IF "DB_McpKeyboardSignals".sK10_LoaderAuto.sKeySWToggleStatus  AND NOT "DB_LoaderOptions".ExtLoadUnload.Disabled THEN
           // Msg: 700820 "Sonplas - Défaut interface de communication"
           "LBP_AlarmMsgs".UserA[08].A70UUxx[20] := NOT #sDiagDPCoupler;

           // Msg: 700821 "Sonplas - Chargeur pas prêt"
           "LBP_AlarmMsgs".UserA[08].A70UUxx[21] := NOT #sReady;

           // Msg: 700822 "Sonplas - Arrêt d'urgence actif"
           "LBP_AlarmMsgs".UserA[08].A70UUxx[22] := #sNoEStop;

           // Msg: 700823 "Sonplas - Porte(s) ouverte(s)"
           "LBP_AlarmMsgs".UserA[08].A70UUxx[23] := NOT #sDoorsClosed;

           // Msg: 700824 "Sonplas - Running error"
           "LBP_AlarmMsgs".UserA[08].A70UUxx[24] := #sRunError;
       ELSE
           "LBP_AlarmMsgs".UserA[08].A70UUxx[20] := FALSE;
           "LBP_AlarmMsgs".UserA[08].A70UUxx[21] := FALSE;
           "LBP_AlarmMsgs".UserA[08].A70UUxx[22] := FALSE;
           "LBP_AlarmMsgs".UserA[08].A70UUxx[23] := FALSE;
           "LBP_AlarmMsgs".UserA[08].A70UUxx[24] := FALSE;
       END_IF;
   END_REGION

   REGION Sonplas Outputs
       REGION Operating_Mode
           // Diagnostic bit DP / DP coupler
           #oOperateOutDiagDPCoupler := FALSE; // WFA A TRAITER

           // Interface partner ready
           #oOperateOutReady := #sAutomaticMode;

           // No emergency stop at Interface partner
           #oOperateOutNoEStop := NOT "DB_DataFromSafety".EmergencyStop;

           // Safety doors closed at Interface partner
           #oOperateOutDoorsClosed := "DB_DataFromSafety".DoorsClosed;

           // Running error
           #oOperateOutRunError := FALSE; // WFA A TRAITER
       END_REGION

       REGION Part Exchange
           // Shuttle 1 in position
           #oPartOutShuttle1InPos := "DB_LoaderShuttle1".sExtLoadUnload.sCurrent_Step_NB = 40
                                  OR "DB_LoaderShuttle1".sExtLoadUnload.sCurrent_Step_NB = 50
                                  OR "DB_LoaderShuttle1".sExtLoadUnload.sCurrent_Step_NB = 70
                                  OR "DB_LoaderShuttle1".sExtLoadUnload.sCurrent_Step_NB = 80
                                  OR "DB_LoaderShuttle1".sExtLoadUnload.sCurrent_Step_NB = 100
                                  OR "DB_LoaderShuttle1".sExtLoadUnload.sCurrent_Step_NB = 110;

           // Part status 1: OK
           #oPartOutPart1OK := "DB_DataPositions".Position[6].FailCode = 0;

           // Part status 1: nOK
           #oPartOutPart1NOK := "DB_DataPositions".Position[6].FailCode <> 0;

           // Shuttle 2 in position
           #oPartOutShuttle2InPos := "DB_LoaderShuttle2".sExtLoadUnload.sCurrent_Step_NB = 40
                                  OR "DB_LoaderShuttle2".sExtLoadUnload.sCurrent_Step_NB = 50
                                  OR "DB_LoaderShuttle2".sExtLoadUnload.sCurrent_Step_NB = 70
                                  OR "DB_LoaderShuttle2".sExtLoadUnload.sCurrent_Step_NB = 80
                                  OR "DB_LoaderShuttle2".sExtLoadUnload.sCurrent_Step_NB = 100
                                  OR "DB_LoaderShuttle2".sExtLoadUnload.sCurrent_Step_NB = 110;

           // Part status 2: OK
           #oPartOutPart2OK := "DB_DataPositions".Position[7].FailCode = 0;

           // Part status 2: nOK
           #oPartOutPart2NOK := "DB_DataPositions".Position[7].FailCode <> 0;
       END_REGION

       REGION Measure
           // Result accepted
           #oMeasureOutResultAccepted := #oMeasureOutResultAccepted;
       END_REGION
   END_REGION
END_FUNCTION_BLOCK

FUNCTION_BLOCK "FB_HmiKeyboardSignals"   // FB810, SCL
{ S7_Optimized_Access := 'TRUE' }
// stored: AutoNumber false, MemoryReserve 100, SetENOAutomatically false
   VAR
      sK1_Powermeter : "FB_HmiKeysSignalsManu";
      sK2_GasAssist { S7_SetPoint := 'True'} : "FB_HmiKeysSignalsManu";
      sK4a_GripperUndrilledPartClose { S7_SetPoint := 'True'} : "FB_HmiKeysSignalsManu";
      sK4b_GripperUndrilledPartOpen { S7_SetPoint := 'True'} : "FB_HmiKeysSignalsManu";
      sK5a_GripperDrilledPartClose { S7_SetPoint := 'True'} : "FB_HmiKeysSignalsManu";
      sK5b_GripperDrilledPartOpen { S7_SetPoint := 'True'} : "FB_HmiKeysSignalsManu";
      sK6_SITestStop { S7_SetPoint := 'True'} : "FB_HmiKeysSignalsManu";
      sK7_FixtureClamp { S7_SetPoint := 'True'} : "FB_HmiKeysSignalsManu";
      sK8_FixtureVacuum { S7_SetPoint := 'True'} : "FB_HmiKeysSignalsManu";
      sK9_Aspiration { S7_SetPoint := 'True'} : "FB_HmiKeysSignalsManu";
      sK12a_Backlight { S7_SetPoint := 'True'} : "FB_HmiKeysSignalsManu";
      sK12b_ObservationCamera { S7_SetPoint := 'True'} : "FB_HmiKeysSignalsManu";
      sK13_MainDoor { S7_SetPoint := 'True'} : "FB_HmiKeysSignalsManu";
      sK14_WarmUp { S7_SetPoint := 'True'} : "FB_HmiKeysSignalsManu";
      sK15_MachineLight { S7_SetPoint := 'True'} : "FB_HmiKeysSignalsManu";
   END_VAR
   VAR_TEMP
      tNoLed : Bool;   // Index for loop
   END_VAR
BEGIN
   REGION Description header 
       //==================================================================================
       // POSALUX Swiss SA / (C) Copyright 2024
       //----------------------------------------------------------------------------------
       // Title: Management of inputs and outputs for HMI buttons
       // Comment/Function: 
       //
       // Author: Fabien WALDT
       // Engineering: TIA Portal v20
       //----------------------------------------------------------------------------------
       // Change log table:
       // Version  | Date     | Expert in charge | Changes applied
       // ---------|----------|------------------|------------------------------------
       // 00.00.01 | 20251024 | WFA              | First released version
       // ==================================================================================
   END_REGION

   REGION HMI Buttons
       // K1_Powermeter 
       #sK1_Powermeter(ioOPC := "DB_OPC_Buttons".Powermeter);

       // K2_GasAssist
       #sK2_GasAssist(ioOPC := "DB_OPC_Buttons".GasAssist);

       // K4_GripperUndrilledPart
       #sK4a_GripperUndrilledPartClose(ioOPC := "DB_OPC_Buttons".GripperUndrilledClamp.Close);
       #sK4b_GripperUndrilledPartOpen(ioOPC := "DB_OPC_Buttons".GripperUndrilledClamp.Open);

       // K5_GripperDrilledPart
       #sK5a_GripperDrilledPartClose(ioOPC := "DB_OPC_Buttons".GripperDrilledClamp.Close);
       #sK5b_GripperDrilledPartOpen(ioOPC := "DB_OPC_Buttons".GripperDrilledClamp.Open);

       // K6_SITestStop
       #sK6_SITestStop(ioOPC := "DB_OPC_Buttons".SITestStop);

       // K7_FixtureClamp
       #sK7_FixtureClamp(ioOPC := "DB_OPC_Buttons".FixtureClamp);

       // K8_FixtureVacuum
       #sK8_FixtureVacuum(ioOPC := "DB_OPC_Buttons".FixtureVacuum);

       // K9_Aspiration
       #sK9_Aspiration(ioOPC := "DB_OPC_Buttons".Aspiration);

       // K12a_Backlight
       #sK12a_Backlight(ioOPC := "DB_OPC_Buttons".Backlight);

       // K12b_ObservationCamera
       #sK12b_ObservationCamera(ioOPC := "DB_OPC_Buttons".ObservationCamera);

       // K13_MainDoor
       #sK13_MainDoor(ioOPC := "DB_OPC_Buttons".MainDoor);

       // K14_WarmUp
       #sK14_WarmUp(ioOPC := "DB_OPC_Buttons".WarmUp);

       // K15_MachineLight
       #sK15_MachineLight(ioOPC := "DB_OPC_Buttons".MachineLight);
   END_REGION

   REGION Gripper
       "DB_OPC_Buttons".GripperUndrilledClamp.IsClosed := "DB_GestionGripper".sUndrilledGripper.oStateCloseWithPart OR "DB_GestionGripper".sUndrilledGripper.oStateClose;
       "DB_OPC_Buttons".GripperUndrilledClamp.IsOpened := "DB_GestionGripper".sUndrilledGripper.oStateOpen;
   END_REGION
END_FUNCTION_BLOCK

FUNCTION_BLOCK "FB_HmiKeysSignalsManu"   // FB813, SCL
{ S7_Optimized_Access := 'TRUE' }
// stored: AutoNumber false, MemoryReserve 100, SetENOAutomatically false
   VAR_IN_OUT
      ioOPC : "UDT_OPC_Button";
   END_VAR
   VAR
      sKeySWStatus : Bool;
      sKeySWToggleStatus : Bool;
      sKeyDisable : Bool;
      sKeySWPositiveFront : Bool;
      sKeySWNegativeFront : Bool;
      sKeySWTogglePositiveFront : Bool;
      sKeySWToggleNegativeFront : Bool;
      sLedSWStatus : Bool;
      sLedSWStatusBlink : Bool;
      sRT_KeySWPositiveFront { S7_SetPoint := 'True'} : R_TRIG;
      sFT_KeySWNegativeFront { S7_SetPoint := 'True'} : F_TRIG;
      sRT_KeySWTogglePositiveFront { S7_SetPoint := 'True'} : R_TRIG;
      sFT_KeySWToggleNegativeFront { S7_SetPoint := 'True'} : F_TRIG;
   END_VAR
BEGIN
   REGION Description header 
       //==================================================================================
       // POSALUX Swiss SA / (C) Copyright 2025
       //----------------------------------------------------------------------------------
       // Title: FB_HmiKeysSignalsManu 
       // Comment/Function: 
       //
       // Author: Fabien Waldt
       // Engineering: TIA Portal v19
       //----------------------------------------------------------------------------------
       // Change log table:
       // Version  | Date     | Expert in charge | Changes applied
       // ---------|----------|------------------|------------------------------------
       // 00.00.01 | 20250911 | WFA              | First released version
       // ==================================================================================
   END_REGION

   REGION Key Enable
       #ioOPC.bEnable := NOT #sKeyDisable;
   END_REGION

   REGION Inputs keys
           // Management of the software input
           IF NOT #sKeyDisable THEN
               #sKeySWStatus := #ioOPC.bClick;
           // ELSE
           //     #sKeySWStatus := FALSE;
           //     #sKeySWToggleStatus := FALSE;
           END_IF;

           // Reset KeyOPCStatus (bClick from HMI)
           #ioOPC.bClick := FALSE;

           // Rising/falling edge detection when pressing the button
           #sRT_KeySWPositiveFront(CLK := #sKeySWStatus,
                                  Q => #sKeySWPositiveFront);

           #sFT_KeySWNegativeFront(CLK := #sKeySWStatus,
                                  Q => #sKeySWNegativeFront);

           // Toggle state update
           IF #sKeySWPositiveFront  THEN
               #sKeySWToggleStatus := NOT #sKeySWToggleStatus;
           END_IF;

           // Rising/falling edge detection of the toggle state
           #sRT_KeySWTogglePositiveFront(CLK := #sKeySWToggleStatus,
                                        Q => #sKeySWTogglePositiveFront);

           #sFT_KeySWToggleNegativeFront(CLK := #sKeySWToggleStatus,
                                        Q => #sKeySWToggleNegativeFront);
   END_REGION

   REGION Outputs LED   
       #ioOPC.bIsPressed := TRUE;

       // On / Off Status
       IF #sLedSWStatus THEN
           #ioOPC.eColor := 2;
       ELSE
           #ioOPC.eColor := 0;
       END_IF;

       // Blink Status
       #ioOPC.bBlink := #sLedSWStatusBlink;
   END_REGION
END_FUNCTION_BLOCK

FUNCTION_BLOCK "FB_Parameters"   // FB64, SCL
{ S7_Optimized_Access := 'TRUE' }
// stored: MemoryReserve 100, SetENOAutomatically false
   VAR
      Shuttle1Enable : "UDT_BoolEnable";
      Shuttle2Enable : Bool;
   END_VAR
   VAR RETAIN
      GazPressureManual : Real := 0.7;   // @Precision:3 @Unit:bar @Min:0.5 @Max:1.2
   END_VAR
   VAR
      CoolingVentilatorSetpoint : Real;
      TemperatureCoolingSetpoint : Real;
      BlowingSetpoint : Real;
      sPresenceShuttle1UndrilledPart : "FB_HMI_PLC_Pos";
      sPresenceShuttle1UndrilledBw { S7_SetPoint := 'True'} : "FB_HMI_PLC_Pos";
      sPresenceShuttle1DrilledPart { S7_SetPoint := 'True'} : "FB_HMI_PLC_Pos";
      sPresenceShuttle1DrilledBw { S7_SetPoint := 'True'} : "FB_HMI_PLC_Pos";
      sPresenceShuttle2UndrilledPart : "FB_HMI_PLC_Pos";
      sPresenceShuttle2UndrilledBw { S7_SetPoint := 'True'} : "FB_HMI_PLC_Pos";
      sPresenceShuttle2DrilledPart { S7_SetPoint := 'True'} : "FB_HMI_PLC_Pos";
      sPresenceShuttle2DrilledBw { S7_SetPoint := 'True'} : "FB_HMI_PLC_Pos";
      sPresenceGripperUndrilledPart : "FB_HMI_PLC_Pos";
      sPresenceGripperUndrilledBw { S7_SetPoint := 'True'} : "FB_HMI_PLC_Pos";
      sPresenceGripperDrilledPart { S7_SetPoint := 'True'} : "FB_HMI_PLC_Pos";
      sPresenceGripperDrilledBw { S7_SetPoint := 'True'} : "FB_HMI_PLC_Pos";
      sPresenceFixtureUndrilledPart : "FB_HMI_PLC_Pos";
      sPresenceFixtureUndrilledBw { S7_SetPoint := 'True'} : "FB_HMI_PLC_Pos";
      sPresenceFixtureDrilledPart { S7_SetPoint := 'True'} : "FB_HMI_PLC_Pos";
      sPresenceFixtureDrilledBw { S7_SetPoint := 'True'} : "FB_HMI_PLC_Pos";
      sHmiChangeEnable { S7_SetPoint := 'True'} : Bool;
   END_VAR
BEGIN
   REGION Description header 
       //==================================================================================
       // POSALUX Swiss SA / (C) Copyright 2025
       //----------------------------------------------------------------------------------
       // Title: FB_OPC_Parameters
       // Comment/Function: 
       // Author: Fabien WALDT
       // Engineering: TIA Portal v20
       //----------------------------------------------------------------------------------
       // Change log table:
       // Version  | Date     | Expert in charge | Changes applied
       // ---------|----------|------------------|-----------------------------------------
       // 00.00.01 | 20260304 | WFA              | First released version
       // =================================================================================
   END_REGION

   REGION Set Points (HMI -> PLC)
       "DB_HMISetting".GasAssistSetPoint := "DB_OPC_Machine".Parameters.GasAssistSetPoint;
       "DB_HMISetting".CoolingVentilatorSetpoint := "DB_OPC_Machine".Parameters.CoolingVentilatorSetpoint;
       "DB_HMISetting".TemperatureCoolingSetpoint := "DB_OPC_Machine".Parameters.TemperatureCoolingSetpoint;
       "DB_HMISetting".BlowingSetpoint := "DB_OPC_Machine".Parameters.BlowingSetpoint;
   END_REGION

   REGION Shuttle Enable (HMI -> PLC)
       "DB_OPC_Machine".Parameters.Shuttle1Enable.IsEnabled := NOT "DB_LoaderShuttle1".sMain.iJobReq AND NOT "DB_LoaderShuttle2".sMain.iJobReq;
       "DB_OPC_Machine".Parameters.Shuttle2Enable.IsEnabled := NOT "DB_LoaderShuttle1".sMain.iJobReq AND NOT "DB_LoaderShuttle2".sMain.iJobReq;

       "DB_HMISetting".Shuttle1Enable := "DB_OPC_Machine".Parameters.Shuttle1Enable.Value;
       "DB_HMISetting".Shuttle2Enable := "DB_OPC_Machine".Parameters.Shuttle2Enable.Value;
   END_REGION

   REGION Sequence
       // Shuttle 1
       "DB_OPC_Machine".Parameters.Sequence.Shuttle1.Main := "DB_LoaderShuttle1".sMain.sCurrent_Step_NB;
       "DB_OPC_Machine".Parameters.Sequence.Shuttle1.ShuttleInt := "DB_LoaderShuttle1".sShuttleInt.sCurrent_Step_NB;
       "DB_OPC_Machine".Parameters.Sequence.Shuttle1.ShuttleExt := "DB_LoaderShuttle1".sShuttleExt.sCurrent_Step_NB;
       "DB_OPC_Machine".Parameters.Sequence.Shuttle1.ControlIn := "DB_LoaderShuttle1".sControlIn.sCurrent_Step_NB;
       "DB_OPC_Machine".Parameters.Sequence.Shuttle1.ControlOut := "DB_LoaderShuttle1".sControlOut.sCurrent_Step_NB;
       "DB_OPC_Machine".Parameters.Sequence.Shuttle1.Blowing := "DB_LoaderShuttle1".sBlowing.sCurrent_Step_NB;
       "DB_OPC_Machine".Parameters.Sequence.Shuttle1.IntLoadUnload := "DB_LoaderShuttle1".sIntLoadUnload.sCurrent_Step_NB;
       "DB_OPC_Machine".Parameters.Sequence.Shuttle1.ExtLoadUnload := "DB_LoaderShuttle1".sExtLoadUnload.sCurrent_Step_NB;
       "DB_OPC_Machine".Parameters.Sequence.Shuttle1.BwLoadUnload := "DB_LoaderShuttle1".sBwLoadUnload.sCurrent_Step_NB;
       "DB_OPC_Machine".Parameters.Sequence.Shuttle1.BwControlIn := "DB_LoaderShuttle1".sBwControlIn.sCurrent_Step_NB;
       "DB_OPC_Machine".Parameters.Sequence.Shuttle1.ActControlIn := "DB_LoaderShuttle1".sActPartControlIn.sCurrent_Step_NB;
       "DB_OPC_Machine".Parameters.Sequence.Shuttle1.ActControlOut := "DB_LoaderShuttle1".sActPartControlOut.sCurrent_Step_NB;
       "DB_OPC_Machine".Parameters.Sequence.Shuttle1.ActBwControlIn := "DB_LoaderShuttle1".sActBwControlIn.sCurrent_Step_NB;

       // Shuttle 2
       "DB_OPC_Machine".Parameters.Sequence.Shuttle2.Main := "DB_LoaderShuttle2".sMain.sCurrent_Step_NB;
       "DB_OPC_Machine".Parameters.Sequence.Shuttle2.ShuttleInt := "DB_LoaderShuttle2".sShuttleInt.sCurrent_Step_NB;
       "DB_OPC_Machine".Parameters.Sequence.Shuttle2.ShuttleExt := "DB_LoaderShuttle2".sShuttleExt.sCurrent_Step_NB;
       "DB_OPC_Machine".Parameters.Sequence.Shuttle2.ControlIn := "DB_LoaderShuttle2".sControlIn.sCurrent_Step_NB;
       "DB_OPC_Machine".Parameters.Sequence.Shuttle2.ControlOut := "DB_LoaderShuttle2".sControlOut.sCurrent_Step_NB;
       "DB_OPC_Machine".Parameters.Sequence.Shuttle2.Blowing := "DB_LoaderShuttle2".sBlowing.sCurrent_Step_NB;
       "DB_OPC_Machine".Parameters.Sequence.Shuttle2.IntLoadUnload := "DB_LoaderShuttle2".sIntLoadUnload.sCurrent_Step_NB;
       "DB_OPC_Machine".Parameters.Sequence.Shuttle2.ExtLoadUnload := "DB_LoaderShuttle2".sExtLoadUnload.sCurrent_Step_NB;
       "DB_OPC_Machine".Parameters.Sequence.Shuttle2.BwLoadUnload := "DB_LoaderShuttle2".sBwLoadUnload.sCurrent_Step_NB;
       "DB_OPC_Machine".Parameters.Sequence.Shuttle2.BwControlIn := "DB_LoaderShuttle2".sBwControlIn.sCurrent_Step_NB;
       "DB_OPC_Machine".Parameters.Sequence.Shuttle2.ActControlIn := "DB_LoaderShuttle2".sActPartControlIn.sCurrent_Step_NB;
       "DB_OPC_Machine".Parameters.Sequence.Shuttle2.ActControlOut := "DB_LoaderShuttle2".sActPartControlout.sCurrent_Step_NB;
       "DB_OPC_Machine".Parameters.Sequence.Shuttle2.ActBwControlIn := "DB_LoaderShuttle2".sActBwControlIn.sCurrent_Step_NB;

       // Fixture
       "DB_OPC_Machine".Parameters.Sequence.Fixture.Blowing := "DB_LoaderFixture".sFixtureBlowing.sCurrent_Step_NB;
       "DB_OPC_Machine".Parameters.Sequence.Fixture.Loading := "DB_LoaderFixture".sFixtureLoading.sCurrent_Step_NB;
       "DB_OPC_Machine".Parameters.Sequence.Fixture.Unloading := "DB_LoaderFixture".sFixtureUnloading.sCurrent_Step_NB;
       "DB_OPC_Machine".Parameters.Sequence.Fixture.V_Init := "DB_LoaderFixture".sFixtureV_Init.sCurrent_Step_NB;
       "DB_OPC_Machine".Parameters.Sequence.Fixture.W_Init := "DB_LoaderFixture".sFixtureW_Init.sCurrent_Step_NB;

   END_REGION

   REGION Presence
       // Shuttle 1
        "DB_OPC_Machine".Parameters.Presence.Shuttle1UndrilledPart := "DB_PartManagement".sPosition.sShuttle1.Undrilled.Presence.Part;
        "DB_OPC_Machine".Parameters.Presence.Shuttle1UndrilledBw := "DB_PartManagement".sPosition.sShuttle1.Undrilled.Presence.BW;
        "DB_OPC_Machine".Parameters.Presence.Shuttle1DrilledPart := "DB_PartManagement".sPosition.sShuttle1.Drilled.Presence.Part;
        "DB_OPC_Machine".Parameters.Presence.Shuttle1DrilledBw := "DB_PartManagement".sPosition.sShuttle1.Drilled.Presence.BW;

